(* IEC 61131-3 sources: open-ot-experiments/st/iec61131/tests, 28 files *)

(* ---- test_authoring_api.st ---- *)
FUNCTION OPENOT_AuthoringHeaderOk : BOOL
VAR_INPUT
    Records : OPENOT_SCAN_RECORD_BUFFER;
    Offset : UINT;
    Length : UINT;
    EventTypeId : UDINT;
    SourceId : UDINT;
END_VAR
VAR
    HeaderOk : BOOL;
    SourceRemaining : UDINT;
    EventRemaining : UDINT;
    Index : UINT;
    Pos : UINT;
END_VAR

HeaderOk :=
    (Length >= UINT#44) AND
    (Records[Offset] = BYTE#16#4F) AND
    (Records[Offset + UINT#1] = BYTE#16#4F) AND
    (Records[Offset + UINT#2] = BYTE#16#54) AND
    (Records[Offset + UINT#3] = BYTE#16#32) AND
    (Records[Offset + UINT#4] = UINT_TO_BYTE(Length MOD UINT#256)) AND
    (Records[Offset + UINT#5] = UINT_TO_BYTE((Length / UINT#256) MOD UINT#256)) AND
    (Records[Offset + UINT#6] = BYTE#16#08) AND
    (Records[Offset + UINT#7] = BYTE#16#00);

SourceRemaining := SourceId;
FOR Index := UINT#0 TO UINT#3 DO
    Pos := Offset + UINT#32 + Index;
    HeaderOk := HeaderOk AND (Records[Pos] = UDINT_TO_BYTE(SourceRemaining MOD UDINT#256));
    SourceRemaining := SourceRemaining / UDINT#256;
END_FOR;

EventRemaining := EventTypeId;
FOR Index := UINT#0 TO UINT#3 DO
    Pos := Offset + UINT#36 + Index;
    HeaderOk := HeaderOk AND (Records[Pos] = UDINT_TO_BYTE(EventRemaining MOD UDINT#256));
    EventRemaining := EventRemaining / UDINT#256;
END_FOR;

OPENOT_AuthoringHeaderOk := HeaderOk;
END_FUNCTION

FUNCTION_BLOCK OPENOT_TestAuthoringApi
VAR_OUTPUT
    Passed : BOOL;
    FirstBatchCount : UINT;
    FirstBatchDelta : ULINT;
    NoChangeCount : UINT;
    NoChangeDelta : ULINT;
    HeadersOk : BOOL;
    EmissionsOk : BOOL;
    ChangeSuppressionOk : BOOL;
END_VAR
VAR
    Producer : OPENOT_Producer;
    BeforeCount : ULINT;
    Offset0 : UINT;
    Offset1 : UINT;
    Offset2 : UINT;
    Length0 : UINT;
    Length1 : UINT;
    Length2 : UINT;
END_VAR

Producer(Execute := FALSE, ResetScanRecords := TRUE);
Producer(Execute := FALSE, ResetScanRecords := FALSE);
BeforeCount := Producer.PublishedRecordCount;
Producer(
    Execute := TRUE,
    Op := UINT#6,
    ValueId := UDINT#2001,
    ValueReal := REAL#12.5,
    DeadbandReal := REAL#0.5,
    HasQuality := FALSE,
    Quality := UINT#0);
Producer(Execute := FALSE, Op := UINT#6);
Producer(
    Execute := TRUE,
    Op := UINT#7,
    ValueId := UDINT#2002,
    ValueInt := DINT#42,
    HasQuality := FALSE,
    Quality := UINT#0);
Producer(Execute := FALSE, Op := UINT#7);
Producer(
    Execute := TRUE,
    Op := UINT#8,
    StateMachineId := UDINT#7,
    Category := UINT#2,
    PreviousState := UINT#0,
    NewState := UINT#1);
Producer(Execute := FALSE, Op := UINT#8);

FirstBatchCount := Producer.ScanRecordCount;
FirstBatchDelta := Producer.PublishedRecordCount - BeforeCount;
Offset0 := Producer.ScanRecordOffsets[0];
Offset1 := Producer.ScanRecordOffsets[1];
Offset2 := Producer.ScanRecordOffsets[2];
Length0 := Producer.ScanRecordLengths[0];
Length1 := Producer.ScanRecordLengths[1];
Length2 := Producer.ScanRecordLengths[2];
HeadersOk :=
    OPENOT_AuthoringHeaderOk(
        Records := Producer.ScanRecords,
        Offset := Offset0,
        Length := Length0,
        EventTypeId := UDINT#16#0002,
        SourceId := UDINT#1) AND
    OPENOT_AuthoringHeaderOk(
        Records := Producer.ScanRecords,
        Offset := Offset1,
        Length := Length1,
        EventTypeId := UDINT#16#0002,
        SourceId := UDINT#1) AND
    OPENOT_AuthoringHeaderOk(
        Records := Producer.ScanRecords,
        Offset := Offset2,
        Length := Length2,
        EventTypeId := UDINT#16#0001,
        SourceId := UDINT#1);

EmissionsOk :=
    (Producer.EmissionCount = UINT#3) AND
    (Producer.Emissions[0].EventTypeId = UDINT#16#0002) AND
    (Producer.Emissions[0].Seq = ULINT#0) AND
    (Producer.Emissions[1].EventTypeId = UDINT#16#0002) AND
    (Producer.Emissions[1].Seq = ULINT#1) AND
    (Producer.Emissions[2].EventTypeId = UDINT#16#0001) AND
    (Producer.Emissions[2].Seq = ULINT#2);

Producer(Execute := FALSE, ResetScanRecords := TRUE);
Producer(Execute := FALSE, ResetScanRecords := FALSE);
BeforeCount := Producer.PublishedRecordCount;
Producer(
    Execute := TRUE,
    Op := UINT#6,
    ValueId := UDINT#2001,
    ValueReal := REAL#12.5,
    DeadbandReal := REAL#0.5,
    HasQuality := FALSE,
    Quality := UINT#0);
Producer(Execute := FALSE, Op := UINT#6);
Producer(
    Execute := TRUE,
    Op := UINT#7,
    ValueId := UDINT#2002,
    ValueInt := DINT#42,
    HasQuality := FALSE,
    Quality := UINT#0);
Producer(Execute := FALSE, Op := UINT#7);
Producer(
    Execute := TRUE,
    Op := UINT#8,
    StateMachineId := UDINT#7,
    Category := UINT#2,
    PreviousState := UINT#0,
    NewState := UINT#1);
Producer(Execute := FALSE, Op := UINT#8);

NoChangeCount := Producer.ScanRecordCount;
NoChangeDelta := Producer.PublishedRecordCount - BeforeCount;
ChangeSuppressionOk := (NoChangeCount = UINT#0) AND (NoChangeDelta = ULINT#0);

Passed :=
    (FirstBatchCount = UINT#3) AND
    (FirstBatchDelta = ULINT#3) AND
    HeadersOk AND
    EmissionsOk AND
    ChangeSuppressionOk;
END_FUNCTION_BLOCK

(* ---- test_conformant_condition_lifecycle.st ---- *)
FUNCTION_BLOCK OPENOT_TestConformantConditionLifecycle
VAR_OUTPUT
    Passed : BOOL;
    AckPassed : BOOL;
    ShelvedPassed : BOOL;
    SuppressedPassed : BOOL;
    OutOfServicePassed : BOOL;
    MismatchIndex : UINT;
END_VAR
VAR
    AckEncoder : OPENOT_EncodeConformantConditionAcknowledged;
    ShelvedEncoder : OPENOT_EncodeConformantConditionShelved;
    SuppressedEncoder : OPENOT_EncodeConformantConditionSuppressed;
    OutOfServiceEncoder : OPENOT_EncodeConformantConditionOutOfService;
    ExpectedAck : ARRAY[0..75] OF BYTE := [
        BYTE#16#4F, BYTE#16#4F, BYTE#16#54, BYTE#16#32, BYTE#16#4C, BYTE#16#00, BYTE#16#08, BYTE#16#00,
        BYTE#16#A0, BYTE#16#CA, BYTE#16#9A, BYTE#16#3B, BYTE#16#00, BYTE#16#00, BYTE#16#00, BYTE#16#00,
        BYTE#16#01, BYTE#16#00, BYTE#16#00, BYTE#16#00, BYTE#16#00, BYTE#16#00, BYTE#16#00, BYTE#16#00,
        BYTE#16#11, BYTE#16#00, BYTE#16#00, BYTE#16#00, BYTE#16#00, BYTE#16#00, BYTE#16#00, BYTE#16#00,
        BYTE#16#42, BYTE#16#00, BYTE#16#00, BYTE#16#00, BYTE#16#02, BYTE#16#02, BYTE#16#00, BYTE#16#00,
        BYTE#16#05, BYTE#16#00, BYTE#16#05, BYTE#16#04, BYTE#16#29, BYTE#16#23, BYTE#16#00, BYTE#16#00,
        BYTE#16#07, BYTE#16#00, BYTE#16#05, BYTE#16#04, BYTE#16#4D, BYTE#16#00, BYTE#16#00, BYTE#16#00,
        BYTE#16#1D, BYTE#16#00, BYTE#16#0C, BYTE#16#0A, BYTE#16#6F, BYTE#16#70, BYTE#16#65, BYTE#16#72,
        BYTE#16#61, BYTE#16#74, BYTE#16#6F, BYTE#16#72, BYTE#16#2D, BYTE#16#61, BYTE#16#00, BYTE#16#00,
        BYTE#16#FA, BYTE#16#EA, BYTE#16#82, BYTE#16#EC
    ];
    ExpectedShelved : ARRAY[0..83] OF BYTE := [
        BYTE#16#4F, BYTE#16#4F, BYTE#16#54, BYTE#16#32, BYTE#16#54, BYTE#16#00, BYTE#16#08, BYTE#16#00,
        BYTE#16#AA, BYTE#16#CA, BYTE#16#9A, BYTE#16#3B, BYTE#16#00, BYTE#16#00, BYTE#16#00, BYTE#16#00,
        BYTE#16#01, BYTE#16#00, BYTE#16#00, BYTE#16#00, BYTE#16#00, BYTE#16#00, BYTE#16#00, BYTE#16#00,
        BYTE#16#12, BYTE#16#00, BYTE#16#00, BYTE#16#00, BYTE#16#00, BYTE#16#00, BYTE#16#00, BYTE#16#00,
        BYTE#16#42, BYTE#16#00, BYTE#16#00, BYTE#16#00, BYTE#16#04, BYTE#16#02, BYTE#16#00, BYTE#16#00,
        BYTE#16#05, BYTE#16#00, BYTE#16#05, BYTE#16#04, BYTE#16#29, BYTE#16#23, BYTE#16#00, BYTE#16#00,
        BYTE#16#07, BYTE#16#00, BYTE#16#05, BYTE#16#04, BYTE#16#4D, BYTE#16#00, BYTE#16#00, BYTE#16#00,
        BYTE#16#1D, BYTE#16#00, BYTE#16#0C, BYTE#16#0A, BYTE#16#6F, BYTE#16#70, BYTE#16#65, BYTE#16#72,
        BYTE#16#61, BYTE#16#74, BYTE#16#6F, BYTE#16#72, BYTE#16#2D, BYTE#16#61, BYTE#16#00, BYTE#16#00,
        BYTE#16#1E, BYTE#16#00, BYTE#16#05, BYTE#16#04, BYTE#16#2C, BYTE#16#01, BYTE#16#00, BYTE#16#00,
        BYTE#16#E5, BYTE#16#3E, BYTE#16#92, BYTE#16#BD
    ];
    ExpectedSuppressed : ARRAY[0..67] OF BYTE := [
        BYTE#16#4F, BYTE#16#4F, BYTE#16#54, BYTE#16#32, BYTE#16#44, BYTE#16#00, BYTE#16#08, BYTE#16#00,
        BYTE#16#B4, BYTE#16#CA, BYTE#16#9A, BYTE#16#3B, BYTE#16#00, BYTE#16#00, BYTE#16#00, BYTE#16#00,
        BYTE#16#01, BYTE#16#00, BYTE#16#00, BYTE#16#00, BYTE#16#00, BYTE#16#00, BYTE#16#00, BYTE#16#00,
        BYTE#16#13, BYTE#16#00, BYTE#16#00, BYTE#16#00, BYTE#16#00, BYTE#16#00, BYTE#16#00, BYTE#16#00,
        BYTE#16#42, BYTE#16#00, BYTE#16#00, BYTE#16#00, BYTE#16#06, BYTE#16#02, BYTE#16#00, BYTE#16#00,
        BYTE#16#05, BYTE#16#00, BYTE#16#05, BYTE#16#04, BYTE#16#29, BYTE#16#23, BYTE#16#00, BYTE#16#00,
        BYTE#16#1F, BYTE#16#00, BYTE#16#0C, BYTE#16#0B, BYTE#16#6D, BYTE#16#61, BYTE#16#69, BYTE#16#6E,
        BYTE#16#74, BYTE#16#65, BYTE#16#6E, BYTE#16#61, BYTE#16#6E, BYTE#16#63, BYTE#16#65, BYTE#16#00,
        BYTE#16#17, BYTE#16#3E, BYTE#16#4F, BYTE#16#63
    ];
    ExpectedOutOfService : ARRAY[0..67] OF BYTE := [
        BYTE#16#4F, BYTE#16#4F, BYTE#16#54, BYTE#16#32, BYTE#16#44, BYTE#16#00, BYTE#16#08, BYTE#16#00,
        BYTE#16#BE, BYTE#16#CA, BYTE#16#9A, BYTE#16#3B, BYTE#16#00, BYTE#16#00, BYTE#16#00, BYTE#16#00,
        BYTE#16#01, BYTE#16#00, BYTE#16#00, BYTE#16#00, BYTE#16#00, BYTE#16#00, BYTE#16#00, BYTE#16#00,
        BYTE#16#14, BYTE#16#00, BYTE#16#00, BYTE#16#00, BYTE#16#00, BYTE#16#00, BYTE#16#00, BYTE#16#00,
        BYTE#16#42, BYTE#16#00, BYTE#16#00, BYTE#16#00, BYTE#16#08, BYTE#16#02, BYTE#16#00, BYTE#16#00,
        BYTE#16#05, BYTE#16#00, BYTE#16#05, BYTE#16#04, BYTE#16#29, BYTE#16#23, BYTE#16#00, BYTE#16#00,
        BYTE#16#1D, BYTE#16#00, BYTE#16#0C, BYTE#16#0A, BYTE#16#6F, BYTE#16#70, BYTE#16#65, BYTE#16#72,
        BYTE#16#61, BYTE#16#74, BYTE#16#6F, BYTE#16#72, BYTE#16#2D, BYTE#16#61, BYTE#16#00, BYTE#16#00,
        BYTE#16#9D, BYTE#16#5C, BYTE#16#A4, BYTE#16#01
    ];
    Index : UINT;
END_VAR

AckEncoder();
ShelvedEncoder();
SuppressedEncoder();
OutOfServiceEncoder();

AckPassed := AckEncoder.Length = UINT#76;
ShelvedPassed := ShelvedEncoder.Length = UINT#84;
SuppressedPassed := SuppressedEncoder.Length = UINT#68;
OutOfServicePassed := OutOfServiceEncoder.Length = UINT#68;
MismatchIndex := UINT#65535;

IF AckPassed THEN
    FOR Index := UINT#0 TO UINT#75 DO
        IF (AckEncoder.Buffer[Index] <> ExpectedAck[Index]) AND (MismatchIndex = UINT#65535) THEN
            AckPassed := FALSE;
            MismatchIndex := Index;
        END_IF;
    END_FOR;
END_IF;

IF ShelvedPassed THEN
    FOR Index := UINT#0 TO UINT#83 DO
        IF (ShelvedEncoder.Buffer[Index] <> ExpectedShelved[Index]) AND (MismatchIndex = UINT#65535) THEN
            ShelvedPassed := FALSE;
            MismatchIndex := Index;
        END_IF;
    END_FOR;
END_IF;

IF SuppressedPassed THEN
    FOR Index := UINT#0 TO UINT#67 DO
        IF (SuppressedEncoder.Buffer[Index] <> ExpectedSuppressed[Index]) AND (MismatchIndex = UINT#65535) THEN
            SuppressedPassed := FALSE;
            MismatchIndex := Index;
        END_IF;
    END_FOR;
END_IF;

IF OutOfServicePassed THEN
    FOR Index := UINT#0 TO UINT#67 DO
        IF (OutOfServiceEncoder.Buffer[Index] <> ExpectedOutOfService[Index]) AND (MismatchIndex = UINT#65535) THEN
            OutOfServicePassed := FALSE;
            MismatchIndex := Index;
        END_IF;
    END_FOR;
END_IF;

Passed := AckPassed AND ShelvedPassed AND SuppressedPassed AND OutOfServicePassed;
END_FUNCTION_BLOCK

(* ---- test_conformant_message.st ---- *)
FUNCTION_BLOCK OPENOT_TestConformantMessage
VAR_OUTPUT
    Passed : BOOL;
    MismatchIndex : UINT;
    ActualLength : UINT;
    ExpectedLength : UINT;
END_VAR
VAR
    Encoder : OPENOT_EncodeConformantMessage;
    Expected : ARRAY[0..75] OF BYTE := [
        BYTE#16#4F, BYTE#16#4F, BYTE#16#54, BYTE#16#32, BYTE#16#4C, BYTE#16#00, BYTE#16#08, BYTE#16#00,
        BYTE#16#0A, BYTE#16#CA, BYTE#16#9A, BYTE#16#3B, BYTE#16#00, BYTE#16#00, BYTE#16#00, BYTE#16#00,
        BYTE#16#01, BYTE#16#00, BYTE#16#00, BYTE#16#00, BYTE#16#00, BYTE#16#00, BYTE#16#00, BYTE#16#00,
        BYTE#16#02, BYTE#16#00, BYTE#16#00, BYTE#16#00, BYTE#16#00, BYTE#16#00, BYTE#16#00, BYTE#16#00,
        BYTE#16#42, BYTE#16#00, BYTE#16#00, BYTE#16#00, BYTE#16#03, BYTE#16#00, BYTE#16#00, BYTE#16#00,
        BYTE#16#14, BYTE#16#00, BYTE#16#05, BYTE#16#04, BYTE#16#E9, BYTE#16#03, BYTE#16#00, BYTE#16#00,
        BYTE#16#15, BYTE#16#00, BYTE#16#0C, BYTE#16#0B, BYTE#16#70, BYTE#16#68, BYTE#16#61, BYTE#16#73,
        BYTE#16#65, BYTE#16#20, BYTE#16#72, BYTE#16#65, BYTE#16#61, BYTE#16#64, BYTE#16#79, BYTE#16#00,
        BYTE#16#08, BYTE#16#00, BYTE#16#03, BYTE#16#02, BYTE#16#F4, BYTE#16#01, BYTE#16#00, BYTE#16#00,
        BYTE#16#CF, BYTE#16#CF, BYTE#16#BE, BYTE#16#B0
    ];
    Index : UINT;
END_VAR

Encoder();
ActualLength := Encoder.Length;
ExpectedLength := UINT#76;
Passed := ActualLength = ExpectedLength;
MismatchIndex := UINT#65535;

IF Passed THEN
    FOR Index := UINT#0 TO ExpectedLength - UINT#1 DO
        IF (Encoder.Buffer[Index] <> Expected[Index]) AND (MismatchIndex = UINT#65535) THEN
            Passed := FALSE;
            MismatchIndex := Index;
        END_IF;
    END_FOR;
END_IF;
END_FUNCTION_BLOCK

(* ---- test_conformant_records_dropped.st ---- *)
FUNCTION_BLOCK OPENOT_TestConformantRecordsDropped
VAR_OUTPUT
    Passed : BOOL;
    MismatchIndex : UINT;
    ActualLength : UINT;
    ExpectedLength : UINT;
END_VAR
VAR
    Encoder : OPENOT_EncodeConformantRecordsDropped;
    Expected : ARRAY[0..99] OF BYTE := [
        BYTE#16#4F, BYTE#16#4F, BYTE#16#54, BYTE#16#32, BYTE#16#64, BYTE#16#00, BYTE#16#08, BYTE#16#00,
        BYTE#16#00, BYTE#16#00, BYTE#16#00, BYTE#16#00, BYTE#16#00, BYTE#16#00, BYTE#16#00, BYTE#16#00,
        BYTE#16#09, BYTE#16#00, BYTE#16#00, BYTE#16#00, BYTE#16#00, BYTE#16#00, BYTE#16#00, BYTE#16#00,
        BYTE#16#64, BYTE#16#00, BYTE#16#00, BYTE#16#00, BYTE#16#00, BYTE#16#00, BYTE#16#00, BYTE#16#00,
        BYTE#16#42, BYTE#16#00, BYTE#16#00, BYTE#16#00, BYTE#16#04, BYTE#16#01, BYTE#16#00, BYTE#16#00,
        BYTE#16#16, BYTE#16#00, BYTE#16#05, BYTE#16#04, BYTE#16#12, BYTE#16#00, BYTE#16#00, BYTE#16#00,
        BYTE#16#17, BYTE#16#00, BYTE#16#07, BYTE#16#08, BYTE#16#28, BYTE#16#00, BYTE#16#00, BYTE#16#00,
        BYTE#16#00, BYTE#16#00, BYTE#16#00, BYTE#16#00, BYTE#16#18, BYTE#16#00, BYTE#16#07, BYTE#16#08,
        BYTE#16#39, BYTE#16#00, BYTE#16#00, BYTE#16#00, BYTE#16#00, BYTE#16#00, BYTE#16#00, BYTE#16#00,
        BYTE#16#19, BYTE#16#00, BYTE#16#0B, BYTE#16#08, BYTE#16#00, BYTE#16#CA, BYTE#16#9A, BYTE#16#3B,
        BYTE#16#00, BYTE#16#00, BYTE#16#00, BYTE#16#00, BYTE#16#1A, BYTE#16#00, BYTE#16#0B, BYTE#16#08,
        BYTE#16#10, BYTE#16#F1, BYTE#16#9A, BYTE#16#3B, BYTE#16#00, BYTE#16#00, BYTE#16#00, BYTE#16#00,
        BYTE#16#09, BYTE#16#8A, BYTE#16#DF, BYTE#16#6D
    ];
    Index : UINT;
END_VAR

Encoder();
ActualLength := Encoder.Length;
ExpectedLength := UINT#100;
Passed := ActualLength = ExpectedLength;
MismatchIndex := UINT#65535;

IF Passed THEN
    FOR Index := UINT#0 TO ExpectedLength - UINT#1 DO
        IF (Encoder.Buffer[Index] <> Expected[Index]) AND (MismatchIndex = UINT#65535) THEN
            Passed := FALSE;
            MismatchIndex := Index;
        END_IF;
    END_FOR;
END_IF;
END_FUNCTION_BLOCK

(* ---- test_conformant_regulated.st ---- *)
FUNCTION_BLOCK OPENOT_TestConformantRegulated
VAR_OUTPUT
    Passed : BOOL;
    OperatorActionPassed : BOOL;
    OperatorLoginPassed : BOOL;
    OperatorLogoutPassed : BOOL;
    SecurityAccessFailurePassed : BOOL;
    ParameterChangeRealPassed : BOOL;
    ParameterChangeIntPassed : BOOL;
    ParameterChangeBitsPassed : BOOL;
    ParameterChangeStringPassed : BOOL;
    MismatchIndex : UINT;
END_VAR
VAR
    OperatorActionEncoder : OPENOT_EncodeConformantOperatorAction;
    OperatorLoginEncoder : OPENOT_EncodeConformantOperatorLogin;
    OperatorLogoutEncoder : OPENOT_EncodeConformantOperatorLogout;
    SecurityAccessFailureEncoder : OPENOT_EncodeConformantSecurityAccessFailure;
    ParameterChangeRealEncoder : OPENOT_EncodeConformantParameterChangeReal;
    ParameterChangeIntEncoder : OPENOT_EncodeConformantParameterChangeInt;
    ParameterChangeBitsEncoder : OPENOT_EncodeConformantParameterChangeBits;
    ParameterChangeStringEncoder : OPENOT_EncodeConformantParameterChangeString;
    ExpectedOperatorAction : ARRAY[0..107] OF BYTE := [
        BYTE#16#4F, BYTE#16#4F, BYTE#16#54, BYTE#16#32, BYTE#16#6C, BYTE#16#00, BYTE#16#08, BYTE#16#00, BYTE#16#36, BYTE#16#CB, BYTE#16#9A, BYTE#16#3B, BYTE#16#00, BYTE#16#00, BYTE#16#00, BYTE#16#00,
        BYTE#16#01, BYTE#16#00, BYTE#16#00, BYTE#16#00, BYTE#16#00, BYTE#16#00, BYTE#16#00, BYTE#16#00, BYTE#16#20, BYTE#16#00, BYTE#16#00, BYTE#16#00, BYTE#16#00, BYTE#16#00, BYTE#16#00, BYTE#16#00,
        BYTE#16#42, BYTE#16#00, BYTE#16#00, BYTE#16#00, BYTE#16#00, BYTE#16#04, BYTE#16#00, BYTE#16#00, BYTE#16#0A, BYTE#16#00, BYTE#16#05, BYTE#16#04, BYTE#16#71, BYTE#16#17, BYTE#16#00, BYTE#16#00,
        BYTE#16#0B, BYTE#16#00, BYTE#16#0C, BYTE#16#0A, BYTE#16#6F, BYTE#16#70, BYTE#16#65, BYTE#16#72, BYTE#16#61, BYTE#16#74, BYTE#16#6F, BYTE#16#72, BYTE#16#2D, BYTE#16#61, BYTE#16#00, BYTE#16#00,
        BYTE#16#0C, BYTE#16#00, BYTE#16#05, BYTE#16#04, BYTE#16#59, BYTE#16#1B, BYTE#16#00, BYTE#16#00, BYTE#16#0C, BYTE#16#00, BYTE#16#05, BYTE#16#04, BYTE#16#5A, BYTE#16#1B, BYTE#16#00, BYTE#16#00,
        BYTE#16#20, BYTE#16#00, BYTE#16#03, BYTE#16#02, BYTE#16#00, BYTE#16#00, BYTE#16#00, BYTE#16#00, BYTE#16#21, BYTE#16#00, BYTE#16#0C, BYTE#16#09, BYTE#16#73, BYTE#16#74, BYTE#16#61, BYTE#16#74,
        BYTE#16#69, BYTE#16#6F, BYTE#16#6E, BYTE#16#2D, BYTE#16#31, BYTE#16#00, BYTE#16#00, BYTE#16#00, BYTE#16#26, BYTE#16#B1, BYTE#16#DF, BYTE#16#49
    ];
    ExpectedOperatorLogin : ARRAY[0..91] OF BYTE := [
        BYTE#16#4F, BYTE#16#4F, BYTE#16#54, BYTE#16#32, BYTE#16#5C, BYTE#16#00, BYTE#16#08, BYTE#16#00, BYTE#16#40, BYTE#16#CB, BYTE#16#9A, BYTE#16#3B, BYTE#16#00, BYTE#16#00, BYTE#16#00, BYTE#16#00,
        BYTE#16#01, BYTE#16#00, BYTE#16#00, BYTE#16#00, BYTE#16#00, BYTE#16#00, BYTE#16#00, BYTE#16#00, BYTE#16#21, BYTE#16#00, BYTE#16#00, BYTE#16#00, BYTE#16#00, BYTE#16#00, BYTE#16#00, BYTE#16#00,
        BYTE#16#42, BYTE#16#00, BYTE#16#00, BYTE#16#00, BYTE#16#01, BYTE#16#04, BYTE#16#00, BYTE#16#00, BYTE#16#0B, BYTE#16#00, BYTE#16#0C, BYTE#16#0A, BYTE#16#6F, BYTE#16#70, BYTE#16#65, BYTE#16#72,
        BYTE#16#61, BYTE#16#74, BYTE#16#6F, BYTE#16#72, BYTE#16#2D, BYTE#16#61, BYTE#16#00, BYTE#16#00, BYTE#16#20, BYTE#16#00, BYTE#16#03, BYTE#16#02, BYTE#16#00, BYTE#16#00, BYTE#16#00, BYTE#16#00,
        BYTE#16#21, BYTE#16#00, BYTE#16#0C, BYTE#16#09, BYTE#16#73, BYTE#16#74, BYTE#16#61, BYTE#16#74, BYTE#16#69, BYTE#16#6F, BYTE#16#6E, BYTE#16#2D, BYTE#16#31, BYTE#16#00, BYTE#16#00, BYTE#16#00,
        BYTE#16#33, BYTE#16#00, BYTE#16#03, BYTE#16#02, BYTE#16#03, BYTE#16#00, BYTE#16#00, BYTE#16#00, BYTE#16#74, BYTE#16#13, BYTE#16#41, BYTE#16#A8
    ];
    ExpectedOperatorLogout : ARRAY[0..75] OF BYTE := [
        BYTE#16#4F, BYTE#16#4F, BYTE#16#54, BYTE#16#32, BYTE#16#4C, BYTE#16#00, BYTE#16#08, BYTE#16#00, BYTE#16#4A, BYTE#16#CB, BYTE#16#9A, BYTE#16#3B, BYTE#16#00, BYTE#16#00, BYTE#16#00, BYTE#16#00,
        BYTE#16#01, BYTE#16#00, BYTE#16#00, BYTE#16#00, BYTE#16#00, BYTE#16#00, BYTE#16#00, BYTE#16#00, BYTE#16#22, BYTE#16#00, BYTE#16#00, BYTE#16#00, BYTE#16#00, BYTE#16#00, BYTE#16#00, BYTE#16#00,
        BYTE#16#42, BYTE#16#00, BYTE#16#00, BYTE#16#00, BYTE#16#02, BYTE#16#04, BYTE#16#00, BYTE#16#00, BYTE#16#0B, BYTE#16#00, BYTE#16#0C, BYTE#16#0A, BYTE#16#6F, BYTE#16#70, BYTE#16#65, BYTE#16#72,
        BYTE#16#61, BYTE#16#74, BYTE#16#6F, BYTE#16#72, BYTE#16#2D, BYTE#16#61, BYTE#16#00, BYTE#16#00, BYTE#16#21, BYTE#16#00, BYTE#16#0C, BYTE#16#09, BYTE#16#73, BYTE#16#74, BYTE#16#61, BYTE#16#74,
        BYTE#16#69, BYTE#16#6F, BYTE#16#6E, BYTE#16#2D, BYTE#16#31, BYTE#16#00, BYTE#16#00, BYTE#16#00, BYTE#16#14, BYTE#16#BF, BYTE#16#E7, BYTE#16#8C
    ];
    ExpectedSecurityAccessFailure : ARRAY[0..87] OF BYTE := [
        BYTE#16#4F, BYTE#16#4F, BYTE#16#54, BYTE#16#32, BYTE#16#58, BYTE#16#00, BYTE#16#08, BYTE#16#00, BYTE#16#54, BYTE#16#CB, BYTE#16#9A, BYTE#16#3B, BYTE#16#00, BYTE#16#00, BYTE#16#00, BYTE#16#00,
        BYTE#16#01, BYTE#16#00, BYTE#16#00, BYTE#16#00, BYTE#16#00, BYTE#16#00, BYTE#16#00, BYTE#16#00, BYTE#16#23, BYTE#16#00, BYTE#16#00, BYTE#16#00, BYTE#16#00, BYTE#16#00, BYTE#16#00, BYTE#16#00,
        BYTE#16#42, BYTE#16#00, BYTE#16#00, BYTE#16#00, BYTE#16#05, BYTE#16#04, BYTE#16#00, BYTE#16#00, BYTE#16#0B, BYTE#16#00, BYTE#16#0C, BYTE#16#0A, BYTE#16#6F, BYTE#16#70, BYTE#16#65, BYTE#16#72,
        BYTE#16#61, BYTE#16#74, BYTE#16#6F, BYTE#16#72, BYTE#16#2D, BYTE#16#78, BYTE#16#00, BYTE#16#00, BYTE#16#21, BYTE#16#00, BYTE#16#0C, BYTE#16#09, BYTE#16#73, BYTE#16#74, BYTE#16#61, BYTE#16#74,
        BYTE#16#69, BYTE#16#6F, BYTE#16#6E, BYTE#16#2D, BYTE#16#32, BYTE#16#00, BYTE#16#00, BYTE#16#00, BYTE#16#1F, BYTE#16#00, BYTE#16#0C, BYTE#16#06, BYTE#16#64, BYTE#16#65, BYTE#16#6E, BYTE#16#69,
        BYTE#16#65, BYTE#16#64, BYTE#16#00, BYTE#16#00, BYTE#16#47, BYTE#16#D1, BYTE#16#30, BYTE#16#F7
    ];
    ExpectedParameterChangeReal : ARRAY[0..111] OF BYTE := [
        BYTE#16#4F, BYTE#16#4F, BYTE#16#54, BYTE#16#32, BYTE#16#70, BYTE#16#00, BYTE#16#08, BYTE#16#00, BYTE#16#5E, BYTE#16#CB, BYTE#16#9A, BYTE#16#3B, BYTE#16#00, BYTE#16#00, BYTE#16#00, BYTE#16#00,
        BYTE#16#01, BYTE#16#00, BYTE#16#00, BYTE#16#00, BYTE#16#00, BYTE#16#00, BYTE#16#00, BYTE#16#00, BYTE#16#24, BYTE#16#00, BYTE#16#00, BYTE#16#00, BYTE#16#00, BYTE#16#00, BYTE#16#00, BYTE#16#00,
        BYTE#16#42, BYTE#16#00, BYTE#16#00, BYTE#16#00, BYTE#16#03, BYTE#16#04, BYTE#16#00, BYTE#16#00, BYTE#16#0D, BYTE#16#00, BYTE#16#05, BYTE#16#04, BYTE#16#D1, BYTE#16#07, BYTE#16#00, BYTE#16#00,
        BYTE#16#0F, BYTE#16#00, BYTE#16#09, BYTE#16#04, BYTE#16#00, BYTE#16#00, BYTE#16#48, BYTE#16#41, BYTE#16#10, BYTE#16#00, BYTE#16#09, BYTE#16#04, BYTE#16#00, BYTE#16#00, BYTE#16#5C, BYTE#16#41,
        BYTE#16#0B, BYTE#16#00, BYTE#16#0C, BYTE#16#0A, BYTE#16#6F, BYTE#16#70, BYTE#16#65, BYTE#16#72, BYTE#16#61, BYTE#16#74, BYTE#16#6F, BYTE#16#72, BYTE#16#2D, BYTE#16#61, BYTE#16#00, BYTE#16#00,
        BYTE#16#1F, BYTE#16#00, BYTE#16#0C, BYTE#16#0F, BYTE#16#73, BYTE#16#65, BYTE#16#74, BYTE#16#70, BYTE#16#6F, BYTE#16#69, BYTE#16#6E, BYTE#16#74, BYTE#16#20, BYTE#16#63, BYTE#16#68, BYTE#16#61,
        BYTE#16#6E, BYTE#16#67, BYTE#16#65, BYTE#16#00, BYTE#16#20, BYTE#16#00, BYTE#16#03, BYTE#16#02, BYTE#16#00, BYTE#16#00, BYTE#16#00, BYTE#16#00, BYTE#16#C6, BYTE#16#34, BYTE#16#40, BYTE#16#11
    ];
    ExpectedParameterChangeInt : ARRAY[0..103] OF BYTE := [
        BYTE#16#4F, BYTE#16#4F, BYTE#16#54, BYTE#16#32, BYTE#16#68, BYTE#16#00, BYTE#16#08, BYTE#16#00, BYTE#16#68, BYTE#16#CB, BYTE#16#9A, BYTE#16#3B, BYTE#16#00, BYTE#16#00, BYTE#16#00, BYTE#16#00,
        BYTE#16#01, BYTE#16#00, BYTE#16#00, BYTE#16#00, BYTE#16#00, BYTE#16#00, BYTE#16#00, BYTE#16#00, BYTE#16#25, BYTE#16#00, BYTE#16#00, BYTE#16#00, BYTE#16#00, BYTE#16#00, BYTE#16#00, BYTE#16#00,
        BYTE#16#42, BYTE#16#00, BYTE#16#00, BYTE#16#00, BYTE#16#03, BYTE#16#04, BYTE#16#00, BYTE#16#00, BYTE#16#0D, BYTE#16#00, BYTE#16#05, BYTE#16#04, BYTE#16#D2, BYTE#16#07, BYTE#16#00, BYTE#16#00,
        BYTE#16#0F, BYTE#16#00, BYTE#16#06, BYTE#16#04, BYTE#16#28, BYTE#16#00, BYTE#16#00, BYTE#16#00, BYTE#16#10, BYTE#16#00, BYTE#16#06, BYTE#16#04, BYTE#16#2A, BYTE#16#00, BYTE#16#00, BYTE#16#00,
        BYTE#16#0B, BYTE#16#00, BYTE#16#0C, BYTE#16#0A, BYTE#16#6F, BYTE#16#70, BYTE#16#65, BYTE#16#72, BYTE#16#61, BYTE#16#74, BYTE#16#6F, BYTE#16#72, BYTE#16#2D, BYTE#16#61, BYTE#16#00, BYTE#16#00,
        BYTE#16#1F, BYTE#16#00, BYTE#16#0C, BYTE#16#0F, BYTE#16#63, BYTE#16#6F, BYTE#16#75, BYTE#16#6E, BYTE#16#74, BYTE#16#20, BYTE#16#63, BYTE#16#6F, BYTE#16#72, BYTE#16#72, BYTE#16#65, BYTE#16#63,
        BYTE#16#74, BYTE#16#65, BYTE#16#64, BYTE#16#00, BYTE#16#7F, BYTE#16#51, BYTE#16#5C, BYTE#16#9A
    ];
    ExpectedParameterChangeBits : ARRAY[0..99] OF BYTE := [
        BYTE#16#4F, BYTE#16#4F, BYTE#16#54, BYTE#16#32, BYTE#16#64, BYTE#16#00, BYTE#16#08, BYTE#16#00, BYTE#16#72, BYTE#16#CB, BYTE#16#9A, BYTE#16#3B, BYTE#16#00, BYTE#16#00, BYTE#16#00, BYTE#16#00,
        BYTE#16#01, BYTE#16#00, BYTE#16#00, BYTE#16#00, BYTE#16#00, BYTE#16#00, BYTE#16#00, BYTE#16#00, BYTE#16#26, BYTE#16#00, BYTE#16#00, BYTE#16#00, BYTE#16#00, BYTE#16#00, BYTE#16#00, BYTE#16#00,
        BYTE#16#42, BYTE#16#00, BYTE#16#00, BYTE#16#00, BYTE#16#03, BYTE#16#04, BYTE#16#00, BYTE#16#00, BYTE#16#0D, BYTE#16#00, BYTE#16#05, BYTE#16#04, BYTE#16#D3, BYTE#16#07, BYTE#16#00, BYTE#16#00,
        BYTE#16#0F, BYTE#16#00, BYTE#16#00, BYTE#16#01, BYTE#16#00, BYTE#16#00, BYTE#16#00, BYTE#16#00, BYTE#16#10, BYTE#16#00, BYTE#16#00, BYTE#16#01, BYTE#16#01, BYTE#16#00, BYTE#16#00, BYTE#16#00,
        BYTE#16#0B, BYTE#16#00, BYTE#16#0C, BYTE#16#0A, BYTE#16#6F, BYTE#16#70, BYTE#16#65, BYTE#16#72, BYTE#16#61, BYTE#16#74, BYTE#16#6F, BYTE#16#72, BYTE#16#2D, BYTE#16#62, BYTE#16#00, BYTE#16#00,
        BYTE#16#1F, BYTE#16#00, BYTE#16#0C, BYTE#16#0C, BYTE#16#65, BYTE#16#6E, BYTE#16#61, BYTE#16#62, BYTE#16#6C, BYTE#16#65, BYTE#16#20, BYTE#16#61, BYTE#16#75, BYTE#16#64, BYTE#16#69, BYTE#16#74,
        BYTE#16#59, BYTE#16#CA, BYTE#16#6A, BYTE#16#6E
    ];
    ExpectedParameterChangeString : ARRAY[0..111] OF BYTE := [
        BYTE#16#4F, BYTE#16#4F, BYTE#16#54, BYTE#16#32, BYTE#16#70, BYTE#16#00, BYTE#16#08, BYTE#16#00, BYTE#16#7C, BYTE#16#CB, BYTE#16#9A, BYTE#16#3B, BYTE#16#00, BYTE#16#00, BYTE#16#00, BYTE#16#00,
        BYTE#16#01, BYTE#16#00, BYTE#16#00, BYTE#16#00, BYTE#16#00, BYTE#16#00, BYTE#16#00, BYTE#16#00, BYTE#16#27, BYTE#16#00, BYTE#16#00, BYTE#16#00, BYTE#16#00, BYTE#16#00, BYTE#16#00, BYTE#16#00,
        BYTE#16#42, BYTE#16#00, BYTE#16#00, BYTE#16#00, BYTE#16#03, BYTE#16#04, BYTE#16#00, BYTE#16#00, BYTE#16#0D, BYTE#16#00, BYTE#16#05, BYTE#16#04, BYTE#16#DC, BYTE#16#07, BYTE#16#00, BYTE#16#00,
        BYTE#16#0F, BYTE#16#00, BYTE#16#0C, BYTE#16#06, BYTE#16#6D, BYTE#16#61, BYTE#16#6E, BYTE#16#75, BYTE#16#61, BYTE#16#6C, BYTE#16#00, BYTE#16#00, BYTE#16#10, BYTE#16#00, BYTE#16#0C, BYTE#16#04,
        BYTE#16#61, BYTE#16#75, BYTE#16#74, BYTE#16#6F, BYTE#16#0B, BYTE#16#00, BYTE#16#0C, BYTE#16#0A, BYTE#16#6F, BYTE#16#70, BYTE#16#65, BYTE#16#72, BYTE#16#61, BYTE#16#74, BYTE#16#6F, BYTE#16#72,
        BYTE#16#2D, BYTE#16#63, BYTE#16#00, BYTE#16#00, BYTE#16#1F, BYTE#16#00, BYTE#16#0C, BYTE#16#09, BYTE#16#6D, BYTE#16#6F, BYTE#16#64, BYTE#16#65, BYTE#16#20, BYTE#16#6E, BYTE#16#6F, BYTE#16#74,
        BYTE#16#65, BYTE#16#00, BYTE#16#00, BYTE#16#00, BYTE#16#20, BYTE#16#00, BYTE#16#03, BYTE#16#02, BYTE#16#01, BYTE#16#00, BYTE#16#00, BYTE#16#00, BYTE#16#76, BYTE#16#BE, BYTE#16#68, BYTE#16#A4
    ];
    Index : UINT;
END_VAR

OperatorActionEncoder();
OperatorLoginEncoder();
OperatorLogoutEncoder();
SecurityAccessFailureEncoder();
ParameterChangeRealEncoder();
ParameterChangeIntEncoder();
ParameterChangeBitsEncoder();
ParameterChangeStringEncoder();

OperatorActionPassed := OperatorActionEncoder.Length = UINT#108;
OperatorLoginPassed := OperatorLoginEncoder.Length = UINT#92;
OperatorLogoutPassed := OperatorLogoutEncoder.Length = UINT#76;
SecurityAccessFailurePassed := SecurityAccessFailureEncoder.Length = UINT#88;
ParameterChangeRealPassed := ParameterChangeRealEncoder.Length = UINT#112;
ParameterChangeIntPassed := ParameterChangeIntEncoder.Length = UINT#104;
ParameterChangeBitsPassed := ParameterChangeBitsEncoder.Length = UINT#100;
ParameterChangeStringPassed := ParameterChangeStringEncoder.Length = UINT#112;
MismatchIndex := UINT#65535;

IF OperatorActionPassed THEN
    FOR Index := UINT#0 TO UINT#107 DO
        IF (OperatorActionEncoder.Buffer[Index] <> ExpectedOperatorAction[Index]) AND (MismatchIndex = UINT#65535) THEN
            OperatorActionPassed := FALSE;
            MismatchIndex := Index;
        END_IF;
    END_FOR;
END_IF;

IF OperatorLoginPassed THEN
    FOR Index := UINT#0 TO UINT#91 DO
        IF (OperatorLoginEncoder.Buffer[Index] <> ExpectedOperatorLogin[Index]) AND (MismatchIndex = UINT#65535) THEN
            OperatorLoginPassed := FALSE;
            MismatchIndex := Index;
        END_IF;
    END_FOR;
END_IF;

IF OperatorLogoutPassed THEN
    FOR Index := UINT#0 TO UINT#75 DO
        IF (OperatorLogoutEncoder.Buffer[Index] <> ExpectedOperatorLogout[Index]) AND (MismatchIndex = UINT#65535) THEN
            OperatorLogoutPassed := FALSE;
            MismatchIndex := Index;
        END_IF;
    END_FOR;
END_IF;

IF SecurityAccessFailurePassed THEN
    FOR Index := UINT#0 TO UINT#87 DO
        IF (SecurityAccessFailureEncoder.Buffer[Index] <> ExpectedSecurityAccessFailure[Index]) AND (MismatchIndex = UINT#65535) THEN
            SecurityAccessFailurePassed := FALSE;
            MismatchIndex := Index;
        END_IF;
    END_FOR;
END_IF;

IF ParameterChangeRealPassed THEN
    FOR Index := UINT#0 TO UINT#111 DO
        IF (ParameterChangeRealEncoder.Buffer[Index] <> ExpectedParameterChangeReal[Index]) AND (MismatchIndex = UINT#65535) THEN
            ParameterChangeRealPassed := FALSE;
            MismatchIndex := Index;
        END_IF;
    END_FOR;
END_IF;

IF ParameterChangeIntPassed THEN
    FOR Index := UINT#0 TO UINT#103 DO
        IF (ParameterChangeIntEncoder.Buffer[Index] <> ExpectedParameterChangeInt[Index]) AND (MismatchIndex = UINT#65535) THEN
            ParameterChangeIntPassed := FALSE;
            MismatchIndex := Index;
        END_IF;
    END_FOR;
END_IF;

IF ParameterChangeBitsPassed THEN
    FOR Index := UINT#0 TO UINT#99 DO
        IF (ParameterChangeBitsEncoder.Buffer[Index] <> ExpectedParameterChangeBits[Index]) AND (MismatchIndex = UINT#65535) THEN
            ParameterChangeBitsPassed := FALSE;
            MismatchIndex := Index;
        END_IF;
    END_FOR;
END_IF;

IF ParameterChangeStringPassed THEN
    FOR Index := UINT#0 TO UINT#111 DO
        IF (ParameterChangeStringEncoder.Buffer[Index] <> ExpectedParameterChangeString[Index]) AND (MismatchIndex = UINT#65535) THEN
            ParameterChangeStringPassed := FALSE;
            MismatchIndex := Index;
        END_IF;
    END_FOR;
END_IF;

Passed := OperatorActionPassed AND OperatorLoginPassed AND OperatorLogoutPassed AND SecurityAccessFailurePassed AND ParameterChangeRealPassed AND ParameterChangeIntPassed AND ParameterChangeBitsPassed AND ParameterChangeStringPassed;
END_FUNCTION_BLOCK

(* ---- test_conformant_source_high_water.st ---- *)
FUNCTION_BLOCK OPENOT_TestConformantSourceHighWater
VAR_OUTPUT
    Passed : BOOL;
    MismatchIndex : UINT;
    ActualLength : UINT;
    ExpectedLength : UINT;
END_VAR
VAR
    Encoder : OPENOT_EncodeConformantSourceHighWater;
    Expected : ARRAY[0..55] OF BYTE := [
        BYTE#16#4F, BYTE#16#4F, BYTE#16#54, BYTE#16#32, BYTE#16#38, BYTE#16#00, BYTE#16#08, BYTE#16#00,
        BYTE#16#00, BYTE#16#00, BYTE#16#00, BYTE#16#00, BYTE#16#00, BYTE#16#00, BYTE#16#00, BYTE#16#00,
        BYTE#16#01, BYTE#16#00, BYTE#16#00, BYTE#16#00, BYTE#16#00, BYTE#16#00, BYTE#16#00, BYTE#16#00,
        BYTE#16#05, BYTE#16#00, BYTE#16#00, BYTE#16#00, BYTE#16#00, BYTE#16#00, BYTE#16#00, BYTE#16#00,
        BYTE#16#58, BYTE#16#00, BYTE#16#00, BYTE#16#00, BYTE#16#08, BYTE#16#01, BYTE#16#00, BYTE#16#80,
        BYTE#16#38, BYTE#16#00, BYTE#16#07, BYTE#16#08, BYTE#16#05, BYTE#16#00, BYTE#16#00, BYTE#16#00,
        BYTE#16#00, BYTE#16#00, BYTE#16#00, BYTE#16#00, BYTE#16#CD, BYTE#16#D4, BYTE#16#74, BYTE#16#86
    ];
    Index : UINT;
END_VAR

Encoder();
ActualLength := Encoder.Length;
ExpectedLength := UINT#56;
Passed := ActualLength = ExpectedLength;
MismatchIndex := UINT#65535;

IF Passed THEN
    FOR Index := UINT#0 TO ExpectedLength - UINT#1 DO
        IF (Encoder.Buffer[Index] <> Expected[Index]) AND (MismatchIndex = UINT#65535) THEN
            Passed := FALSE;
            MismatchIndex := Index;
        END_IF;
    END_FOR;
END_IF;
END_FUNCTION_BLOCK

(* ---- test_conformant_state_transition.st ---- *)
FUNCTION_BLOCK OPENOT_TestConformantStateTransition
VAR_OUTPUT
    Passed : BOOL;
    MismatchIndex : UINT;
    ActualLength : UINT;
    ExpectedLength : UINT;
END_VAR
VAR
    Encoder : OPENOT_EncodeConformantStateTransition;
    Expected : ARRAY[0..75] OF BYTE := [
        BYTE#16#4F, BYTE#16#4F, BYTE#16#54, BYTE#16#32, BYTE#16#4C, BYTE#16#00, BYTE#16#08, BYTE#16#00,
        BYTE#16#00, BYTE#16#CA, BYTE#16#9A, BYTE#16#3B, BYTE#16#00, BYTE#16#00, BYTE#16#00, BYTE#16#00,
        BYTE#16#01, BYTE#16#00, BYTE#16#00, BYTE#16#00, BYTE#16#00, BYTE#16#00, BYTE#16#00, BYTE#16#00,
        BYTE#16#01, BYTE#16#00, BYTE#16#00, BYTE#16#00, BYTE#16#00, BYTE#16#00, BYTE#16#00, BYTE#16#00,
        BYTE#16#42, BYTE#16#00, BYTE#16#00, BYTE#16#00, BYTE#16#01, BYTE#16#00, BYTE#16#00, BYTE#16#00,
        BYTE#16#01, BYTE#16#00, BYTE#16#05, BYTE#16#04, BYTE#16#07, BYTE#16#00, BYTE#16#00, BYTE#16#00,
        BYTE#16#02, BYTE#16#00, BYTE#16#03, BYTE#16#02, BYTE#16#02, BYTE#16#00, BYTE#16#00, BYTE#16#00,
        BYTE#16#03, BYTE#16#00, BYTE#16#03, BYTE#16#02, BYTE#16#03, BYTE#16#00, BYTE#16#00, BYTE#16#00,
        BYTE#16#04, BYTE#16#00, BYTE#16#03, BYTE#16#02, BYTE#16#04, BYTE#16#00, BYTE#16#00, BYTE#16#00,
        BYTE#16#60, BYTE#16#A3, BYTE#16#A5, BYTE#16#47
    ];
    Index : UINT;
END_VAR

Encoder();
ActualLength := Encoder.Length;
ExpectedLength := UINT#76;
Passed := ActualLength = ExpectedLength;
MismatchIndex := UINT#65535;

IF Passed THEN
    FOR Index := UINT#0 TO ExpectedLength - UINT#1 DO
        IF (Encoder.Buffer[Index] <> Expected[Index]) AND (MismatchIndex = UINT#65535) THEN
            Passed := FALSE;
            MismatchIndex := Index;
        END_IF;
    END_FOR;
END_IF;
END_FUNCTION_BLOCK

(* ---- test_conformant_value_changed_int.st ---- *)
FUNCTION_BLOCK OPENOT_TestConformantValueChangedInt
VAR_OUTPUT
    Passed : BOOL;
    MismatchIndex : UINT;
    ActualLength : UINT;
    ExpectedLength : UINT;
END_VAR
VAR
    Encoder : OPENOT_EncodeValueChangedInt;
    Expected : ARRAY[0..75] OF BYTE := [
        BYTE#16#4F, BYTE#16#4F, BYTE#16#54, BYTE#16#32, BYTE#16#4C, BYTE#16#00, BYTE#16#08, BYTE#16#00,
        BYTE#16#1E, BYTE#16#CA, BYTE#16#9A, BYTE#16#3B, BYTE#16#00, BYTE#16#00, BYTE#16#00, BYTE#16#00,
        BYTE#16#01, BYTE#16#00, BYTE#16#00, BYTE#16#00, BYTE#16#00, BYTE#16#00, BYTE#16#00, BYTE#16#00,
        BYTE#16#04, BYTE#16#00, BYTE#16#00, BYTE#16#00, BYTE#16#00, BYTE#16#00, BYTE#16#00, BYTE#16#00,
        BYTE#16#42, BYTE#16#00, BYTE#16#00, BYTE#16#00, BYTE#16#02, BYTE#16#00, BYTE#16#00, BYTE#16#00,
        BYTE#16#0D, BYTE#16#00, BYTE#16#05, BYTE#16#04, BYTE#16#D2, BYTE#16#07, BYTE#16#00, BYTE#16#00,
        BYTE#16#0F, BYTE#16#00, BYTE#16#06, BYTE#16#04, BYTE#16#28, BYTE#16#00, BYTE#16#00, BYTE#16#00,
        BYTE#16#10, BYTE#16#00, BYTE#16#06, BYTE#16#04, BYTE#16#2A, BYTE#16#00, BYTE#16#00, BYTE#16#00,
        BYTE#16#11, BYTE#16#00, BYTE#16#03, BYTE#16#02, BYTE#16#00, BYTE#16#00, BYTE#16#00, BYTE#16#00,
        BYTE#16#A1, BYTE#16#BB, BYTE#16#E9, BYTE#16#2E
    ];
    Index : UINT;
END_VAR

Encoder(
    SourceId := UDINT#66,
    RunId := ULINT#1,
    Seq := ULINT#4,
    SourceTime := ULINT#1000000030,
    ValueId := UDINT#2002,
    NewValue := DINT#42,
    HasPrevious := TRUE,
    PreviousValue := DINT#40,
    HasQuality := TRUE,
    Quality := UINT#0);
ActualLength := Encoder.Length;
ExpectedLength := UINT#76;
Passed := ActualLength = ExpectedLength;
MismatchIndex := UINT#65535;

IF Passed THEN
    FOR Index := UINT#0 TO ExpectedLength - UINT#1 DO
        IF (Encoder.Buffer[Index] <> Expected[Index]) AND (MismatchIndex = UINT#65535) THEN
            Passed := FALSE;
            MismatchIndex := Index;
        END_IF;
    END_FOR;
END_IF;
END_FUNCTION_BLOCK

(* ---- test_control_block.st ---- *)
FUNCTION_BLOCK OPENOT_TestControlBlock
VAR_OUTPUT
    Passed : BOOL;
    MismatchIndex : UINT;
    ActualLength : UINT;
    ExpectedLength : UINT;
END_VAR
VAR
    Writer : OPENOT_WriteControlBlockFixture;
    Expected : ARRAY[0..87] OF BYTE := [
        BYTE#16#4F, BYTE#16#4F, BYTE#16#54, BYTE#16#32, BYTE#16#02, BYTE#16#03, BYTE#16#00, BYTE#16#00,
        BYTE#16#07, BYTE#16#00, BYTE#16#00, BYTE#16#00, BYTE#16#00, BYTE#16#10, BYTE#16#00, BYTE#16#00,
        BYTE#16#02, BYTE#16#00, BYTE#16#00, BYTE#16#00, BYTE#16#00, BYTE#16#00, BYTE#16#00, BYTE#16#00,
        BYTE#16#00, BYTE#16#20, BYTE#16#00, BYTE#16#00, BYTE#16#00, BYTE#16#00, BYTE#16#00, BYTE#16#00,
        BYTE#16#00, BYTE#16#18, BYTE#16#00, BYTE#16#00, BYTE#16#00, BYTE#16#00, BYTE#16#00, BYTE#16#00,
        BYTE#16#0C, BYTE#16#00, BYTE#16#00, BYTE#16#00, BYTE#16#00, BYTE#16#00, BYTE#16#00, BYTE#16#00,
        BYTE#16#03, BYTE#16#00, BYTE#16#00, BYTE#16#00, BYTE#16#00, BYTE#16#00, BYTE#16#00, BYTE#16#00,
        BYTE#16#05, BYTE#16#00, BYTE#16#00, BYTE#16#00, BYTE#16#00, BYTE#16#00, BYTE#16#00, BYTE#16#00,
        BYTE#16#58, BYTE#16#1B, BYTE#16#00, BYTE#16#00, BYTE#16#00, BYTE#16#00, BYTE#16#00, BYTE#16#00,
        BYTE#16#64, BYTE#16#65, BYTE#16#66, BYTE#16#68, BYTE#16#61, BYTE#16#73, BYTE#16#68, BYTE#16#31,
        BYTE#16#6F, BYTE#16#6C, BYTE#16#64, BYTE#16#68, BYTE#16#61, BYTE#16#73, BYTE#16#68, BYTE#16#31
    ];
    Index : UINT;
END_VAR

Writer();
ActualLength := Writer.Length;
ExpectedLength := UINT#88;
Passed := ActualLength = ExpectedLength;
MismatchIndex := UINT#65535;

IF Passed THEN
    FOR Index := UINT#0 TO ExpectedLength - UINT#1 DO
        IF (Writer.Buffer[Index] <> Expected[Index]) AND (MismatchIndex = UINT#65535) THEN
            Passed := FALSE;
            MismatchIndex := Index;
        END_IF;
    END_FOR;
END_IF;
END_FUNCTION_BLOCK

(* ---- test_crc32c_kat.st ---- *)
FUNCTION_BLOCK OPENOT_TestCrc32cKat
VAR_OUTPUT
    Passed : BOOL;
    MismatchIndex : UINT;
    ActualLength : UINT;
    ExpectedLength : UINT;
    ActualCrc : DWORD;
    ExpectedCrc : DWORD;
END_VAR
VAR
    Data : OPENOT_BYTE_BUFFER;
END_VAR

Data[0] := BYTE#16#31;
Data[1] := BYTE#16#32;
Data[2] := BYTE#16#33;
Data[3] := BYTE#16#34;
Data[4] := BYTE#16#35;
Data[5] := BYTE#16#36;
Data[6] := BYTE#16#37;
Data[7] := BYTE#16#38;
Data[8] := BYTE#16#39;

ActualLength := UINT#9;
ExpectedLength := UINT#9;
ActualCrc := OPENOT_Crc32c(Data := Data, Length := UINT#9);
ExpectedCrc := DWORD#16#E3069283;
Passed := ActualCrc = ExpectedCrc;

IF Passed THEN
    MismatchIndex := UINT#65535;
ELSE
    MismatchIndex := UINT#0;
END_IF;
END_FUNCTION_BLOCK

(* ---- test_definition_changed.st ---- *)
FUNCTION_BLOCK OPENOT_TestDefinitionChanged
VAR_OUTPUT
    Passed : BOOL;
    MismatchIndex : UINT;
    ActualLength : UINT;
    ExpectedLength : UINT;
END_VAR
VAR
    Encoder : OPENOT_EncodeDefinitionChanged;
    DefHashOld : OPENOT_HASH8 := [
        BYTE#16#6F, BYTE#16#6C, BYTE#16#64, BYTE#16#68,
        BYTE#16#61, BYTE#16#73, BYTE#16#68, BYTE#16#31
    ];
    DefHashNew : OPENOT_HASH8 := [
        BYTE#16#6E, BYTE#16#65, BYTE#16#77, BYTE#16#68,
        BYTE#16#61, BYTE#16#73, BYTE#16#68, BYTE#16#32
    ];
    Expected : ARRAY[0..79] OF BYTE := [
        BYTE#16#4F, BYTE#16#4F, BYTE#16#54, BYTE#16#32, BYTE#16#50, BYTE#16#00, BYTE#16#08, BYTE#16#00,
        BYTE#16#00, BYTE#16#00, BYTE#16#00, BYTE#16#00, BYTE#16#00, BYTE#16#00, BYTE#16#00, BYTE#16#00,
        BYTE#16#01, BYTE#16#00, BYTE#16#00, BYTE#16#00, BYTE#16#00, BYTE#16#00, BYTE#16#00, BYTE#16#00,
        BYTE#16#01, BYTE#16#00, BYTE#16#00, BYTE#16#00, BYTE#16#00, BYTE#16#00, BYTE#16#00, BYTE#16#00,
        BYTE#16#00, BYTE#16#00, BYTE#16#00, BYTE#16#00, BYTE#16#06, BYTE#16#01, BYTE#16#00, BYTE#16#00,
        BYTE#16#39, BYTE#16#00, BYTE#16#0D, BYTE#16#08, BYTE#16#6F, BYTE#16#6C, BYTE#16#64, BYTE#16#68,
        BYTE#16#61, BYTE#16#73, BYTE#16#68, BYTE#16#31, BYTE#16#1C, BYTE#16#00, BYTE#16#0D, BYTE#16#08,
        BYTE#16#6E, BYTE#16#65, BYTE#16#77, BYTE#16#68, BYTE#16#61, BYTE#16#73, BYTE#16#68, BYTE#16#32,
        BYTE#16#3A, BYTE#16#00, BYTE#16#07, BYTE#16#08, BYTE#16#02, BYTE#16#00, BYTE#16#00, BYTE#16#00,
        BYTE#16#00, BYTE#16#00, BYTE#16#00, BYTE#16#00, BYTE#16#A5, BYTE#16#41, BYTE#16#2E, BYTE#16#B1
    ];
    Index : UINT;
END_VAR

Encoder(
    RunId := ULINT#1,
    Seq := ULINT#1,
    DefHashOld := DefHashOld,
    DefHashNew := DefHashNew,
    EpochId := ULINT#2,
    SourceTime := ULINT#0);
ActualLength := Encoder.Length;
ExpectedLength := UINT#80;
Passed := ActualLength = ExpectedLength;
MismatchIndex := UINT#65535;

IF Passed THEN
    FOR Index := UINT#0 TO ExpectedLength - UINT#1 DO
        IF (Encoder.Buffer[Index] <> Expected[Index]) AND (MismatchIndex = UINT#65535) THEN
            Passed := FALSE;
            MismatchIndex := Index;
        END_IF;
    END_FOR;
END_IF;
END_FUNCTION_BLOCK

(* ---- test_logger_started_cold.st ---- *)
FUNCTION_BLOCK OPENOT_TestLoggerStartedCold
VAR_OUTPUT
    Passed : BOOL;
    MismatchIndex : UINT;
    ActualLength : UINT;
    ExpectedLength : UINT;
END_VAR
VAR
    Encoder : OPENOT_EncodeLoggerStarted;
    Expected : ARRAY[0..51] OF BYTE := [
        BYTE#16#4F, BYTE#16#4F, BYTE#16#54, BYTE#16#32, BYTE#16#34, BYTE#16#00, BYTE#16#08, BYTE#16#00,
        BYTE#16#00, BYTE#16#00, BYTE#16#00, BYTE#16#00, BYTE#16#00, BYTE#16#00, BYTE#16#00, BYTE#16#00,
        BYTE#16#02, BYTE#16#00, BYTE#16#00, BYTE#16#00, BYTE#16#00, BYTE#16#00, BYTE#16#00, BYTE#16#00,
        BYTE#16#00, BYTE#16#00, BYTE#16#00, BYTE#16#00, BYTE#16#00, BYTE#16#00, BYTE#16#00, BYTE#16#00,
        BYTE#16#00, BYTE#16#00, BYTE#16#00, BYTE#16#00, BYTE#16#01, BYTE#16#01, BYTE#16#00, BYTE#16#00,
        BYTE#16#3B, BYTE#16#00, BYTE#16#00, BYTE#16#01, BYTE#16#01, BYTE#16#00, BYTE#16#00, BYTE#16#00,
        BYTE#16#CF, BYTE#16#2A, BYTE#16#DF, BYTE#16#09
    ];
    Index : UINT;
END_VAR

Encoder(RunId := ULINT#2, Seq := ULINT#0, ColdStart := TRUE, SourceTime := ULINT#0);
ActualLength := Encoder.Length;
ExpectedLength := UINT#52;
Passed := ActualLength = ExpectedLength;
MismatchIndex := UINT#65535;

IF Passed THEN
    FOR Index := UINT#0 TO ExpectedLength - UINT#1 DO
        IF (Encoder.Buffer[Index] <> Expected[Index]) AND (MismatchIndex = UINT#65535) THEN
            Passed := FALSE;
            MismatchIndex := Index;
        END_IF;
    END_FOR;
END_IF;
END_FUNCTION_BLOCK

(* ---- test_logger_started_warm.st ---- *)
FUNCTION_BLOCK OPENOT_TestLoggerStartedWarm
VAR_OUTPUT
    Passed : BOOL;
    MismatchIndex : UINT;
    ActualLength : UINT;
    ExpectedLength : UINT;
END_VAR
VAR
    Encoder : OPENOT_EncodeLoggerStarted;
    Expected : ARRAY[0..51] OF BYTE := [
        BYTE#16#4F, BYTE#16#4F, BYTE#16#54, BYTE#16#32, BYTE#16#34, BYTE#16#00, BYTE#16#08, BYTE#16#00,
        BYTE#16#00, BYTE#16#00, BYTE#16#00, BYTE#16#00, BYTE#16#00, BYTE#16#00, BYTE#16#00, BYTE#16#00,
        BYTE#16#01, BYTE#16#00, BYTE#16#00, BYTE#16#00, BYTE#16#00, BYTE#16#00, BYTE#16#00, BYTE#16#00,
        BYTE#16#02, BYTE#16#00, BYTE#16#00, BYTE#16#00, BYTE#16#00, BYTE#16#00, BYTE#16#00, BYTE#16#00,
        BYTE#16#00, BYTE#16#00, BYTE#16#00, BYTE#16#00, BYTE#16#01, BYTE#16#01, BYTE#16#00, BYTE#16#00,
        BYTE#16#3B, BYTE#16#00, BYTE#16#00, BYTE#16#01, BYTE#16#00, BYTE#16#00, BYTE#16#00, BYTE#16#00,
        BYTE#16#C7, BYTE#16#02, BYTE#16#02, BYTE#16#E3
    ];
    Index : UINT;
END_VAR

Encoder(RunId := ULINT#1, Seq := ULINT#2, ColdStart := FALSE, SourceTime := ULINT#0);
ActualLength := Encoder.Length;
ExpectedLength := UINT#52;
Passed := ActualLength = ExpectedLength;
MismatchIndex := UINT#65535;

IF Passed THEN
    FOR Index := UINT#0 TO ExpectedLength - UINT#1 DO
        IF (Encoder.Buffer[Index] <> Expected[Index]) AND (MismatchIndex = UINT#65535) THEN
            Passed := FALSE;
            MismatchIndex := Index;
        END_IF;
    END_FOR;
END_IF;
END_FUNCTION_BLOCK

(* ---- test_logger_stopped.st ---- *)
FUNCTION_BLOCK OPENOT_TestLoggerStopped
VAR_OUTPUT
    Passed : BOOL;
    MismatchIndex : UINT;
    ActualLength : UINT;
    ExpectedLength : UINT;
END_VAR
VAR
    Encoder : OPENOT_EncodeLoggerStopped;
    Expected : ARRAY[0..43] OF BYTE := [
        BYTE#16#4F, BYTE#16#4F, BYTE#16#54, BYTE#16#32, BYTE#16#2C, BYTE#16#00, BYTE#16#08, BYTE#16#00,
        BYTE#16#00, BYTE#16#00, BYTE#16#00, BYTE#16#00, BYTE#16#00, BYTE#16#00, BYTE#16#00, BYTE#16#00,
        BYTE#16#01, BYTE#16#00, BYTE#16#00, BYTE#16#00, BYTE#16#00, BYTE#16#00, BYTE#16#00, BYTE#16#00,
        BYTE#16#00, BYTE#16#00, BYTE#16#00, BYTE#16#00, BYTE#16#00, BYTE#16#00, BYTE#16#00, BYTE#16#00,
        BYTE#16#00, BYTE#16#00, BYTE#16#00, BYTE#16#00, BYTE#16#02, BYTE#16#01, BYTE#16#00, BYTE#16#00,
        BYTE#16#09, BYTE#16#A8, BYTE#16#70, BYTE#16#85
    ];
    Index : UINT;
END_VAR

Encoder(RunId := ULINT#1, Seq := ULINT#0, SourceTime := ULINT#0);
ActualLength := Encoder.Length;
ExpectedLength := UINT#44;
Passed := ActualLength = ExpectedLength;
MismatchIndex := UINT#65535;

IF Passed THEN
    FOR Index := UINT#0 TO ExpectedLength - UINT#1 DO
        IF (Encoder.Buffer[Index] <> Expected[Index]) AND (MismatchIndex = UINT#65535) THEN
            Passed := FALSE;
            MismatchIndex := Index;
        END_IF;
    END_FOR;
END_IF;
END_FUNCTION_BLOCK

(* ---- test_loss_range_formation.st ---- *)
FUNCTION_BLOCK OPENOT_EncodeFormationMinimalMessage
VAR_INPUT
    SourceId : UDINT;
    Seq : ULINT;
END_VAR
VAR_OUTPUT
    Buffer : OPENOT_BYTE_BUFFER;
    Length : UINT;
END_VAR
VAR
    Pos : UINT;
    Crc : DWORD;
END_VAR

Pos := OPENOT_WriteHeader(
    TotalLength := UINT#44,
    Flags := UINT#16#0008,
    SourceTime := ULINT#1780000000000000000 + Seq,
    RunId := ULINT#1,
    Seq := Seq,
    SourceId := SourceId,
    EventTypeId := UDINT#16#0003,
    Buffer := Buffer);

Crc := OPENOT_Crc32c(Data := Buffer, Length := Pos);
Pos := OPENOT_WriteDWordLE(Offset := Pos, Value := Crc, Buffer := Buffer);
Length := Pos;
END_FUNCTION_BLOCK

FUNCTION_BLOCK OPENOT_TestLossRangeFormation
VAR_OUTPUT
    Passed : BOOL;
    FoundSource : BOOL;
    ActualFirstSeq : ULINT;
    ActualLastSeq : ULINT;
    ActualCount : ULINT;
    ActualLossRangeCount : UINT;
    ActualLostCount : ULINT;
END_VAR
VAR
    Producer : OPENOT_Ring256Producer;
    Encoder : OPENOT_EncodeFormationMinimalMessage;
    SeqIndex : UINT;
    LossIndex : UINT;
    SeqValue : ULINT;
    Ran : BOOL;
END_VAR

IF NOT Ran THEN
    FOR SeqIndex := UINT#0 TO UINT#4 DO
        SeqValue := UINT_TO_ULINT(SeqIndex);
        Encoder(SourceId := UDINT#88, Seq := SeqValue);
        Producer(
            Execute := TRUE,
            Record := Encoder.Buffer,
            Length := Encoder.Length,
            RunId := ULINT#1,
            SourceId := UDINT#88,
            Seq := SeqValue);
    END_FOR;

    FOR SeqIndex := UINT#0 TO UINT#79 DO
        SeqValue := UINT_TO_ULINT(SeqIndex);
        Encoder(SourceId := UDINT#99, Seq := SeqValue);
        Producer(
            Execute := TRUE,
            Record := Encoder.Buffer,
            Length := Encoder.Length,
            RunId := ULINT#1,
            SourceId := UDINT#99,
            Seq := SeqValue);
    END_FOR;

    Ran := TRUE;
END_IF;

FoundSource := FALSE;
ActualFirstSeq := ULINT#0;
ActualLastSeq := ULINT#0;
ActualCount := ULINT#0;
ActualLossRangeCount := Producer.LossRangeCount;
ActualLostCount := Producer.LostCount;

IF Producer.LossRangeCount > UINT#0 THEN
    FOR LossIndex := UINT#0 TO Producer.LossRangeCount - UINT#1 DO
        IF (Producer.LossRanges[LossIndex].RunId = ULINT#1) AND (Producer.LossRanges[LossIndex].SourceId = UDINT#88) AND (NOT FoundSource) THEN
            FoundSource := TRUE;
            ActualFirstSeq := Producer.LossRanges[LossIndex].FirstSeq;
            ActualLastSeq := Producer.LossRanges[LossIndex].LastSeq;
            ActualCount := (ActualLastSeq - ActualFirstSeq) + ULINT#1;
        END_IF;
    END_FOR;
END_IF;

Passed :=
    FoundSource AND
    (ActualFirstSeq = ULINT#0) AND
    (ActualLastSeq = ULINT#4) AND
    (ActualCount = ULINT#5) AND
    (NOT Producer.LossRangeOverflow) AND
    (NOT Producer.Error);
END_FUNCTION_BLOCK

(* ---- test_loss_range_interleaved.st ---- *)
FUNCTION_BLOCK OPENOT_EncodeInterleavedMinimalMessage
VAR_INPUT
    SourceId : UDINT;
    Seq : ULINT;
END_VAR
VAR_OUTPUT
    Buffer : OPENOT_BYTE_BUFFER;
    Length : UINT;
END_VAR
VAR
    Pos : UINT;
    Crc : DWORD;
END_VAR

Pos := OPENOT_WriteHeader(
    TotalLength := UINT#44,
    Flags := UINT#16#0008,
    SourceTime := ULINT#1780000000000000000 + Seq,
    RunId := ULINT#1,
    Seq := Seq,
    SourceId := SourceId,
    EventTypeId := UDINT#16#0003,
    Buffer := Buffer);

Crc := OPENOT_Crc32c(Data := Buffer, Length := Pos);
Pos := OPENOT_WriteDWordLE(Offset := Pos, Value := Crc, Buffer := Buffer);
Length := Pos;
END_FUNCTION_BLOCK

FUNCTION_BLOCK OPENOT_TestLossRangeInterleaved
VAR_OUTPUT
    Passed : BOOL;
    ActualLossRangeCount : UINT;
    ActualLostCount : ULINT;
END_VAR
VAR
    Producer : OPENOT_Ring256Producer;
    Encoder : OPENOT_EncodeInterleavedMinimalMessage;
    Ran : BOOL;
END_VAR

IF NOT Ran THEN
    Encoder(SourceId := UDINT#10, Seq := ULINT#0);
    Producer(
        Execute := TRUE,
        Record := Encoder.Buffer,
        Length := Encoder.Length,
        RunId := ULINT#1,
        SourceId := UDINT#10,
        Seq := ULINT#0);
    Encoder(SourceId := UDINT#20, Seq := ULINT#0);
    Producer(
        Execute := TRUE,
        Record := Encoder.Buffer,
        Length := Encoder.Length,
        RunId := ULINT#1,
        SourceId := UDINT#20,
        Seq := ULINT#0);
    Encoder(SourceId := UDINT#10, Seq := ULINT#1);
    Producer(
        Execute := TRUE,
        Record := Encoder.Buffer,
        Length := Encoder.Length,
        RunId := ULINT#1,
        SourceId := UDINT#10,
        Seq := ULINT#1);
    Encoder(SourceId := UDINT#20, Seq := ULINT#1);
    Producer(
        Execute := TRUE,
        Record := Encoder.Buffer,
        Length := Encoder.Length,
        RunId := ULINT#1,
        SourceId := UDINT#20,
        Seq := ULINT#1);
    Encoder(SourceId := UDINT#10, Seq := ULINT#2);
    Producer(
        Execute := TRUE,
        Record := Encoder.Buffer,
        Length := Encoder.Length,
        RunId := ULINT#1,
        SourceId := UDINT#10,
        Seq := ULINT#2);
    Encoder(SourceId := UDINT#20, Seq := ULINT#2);
    Producer(
        Execute := TRUE,
        Record := Encoder.Buffer,
        Length := Encoder.Length,
        RunId := ULINT#1,
        SourceId := UDINT#20,
        Seq := ULINT#2);
    Encoder(SourceId := UDINT#10, Seq := ULINT#3);
    Producer(
        Execute := TRUE,
        Record := Encoder.Buffer,
        Length := Encoder.Length,
        RunId := ULINT#1,
        SourceId := UDINT#10,
        Seq := ULINT#3);
    Encoder(SourceId := UDINT#20, Seq := ULINT#3);
    Producer(
        Execute := TRUE,
        Record := Encoder.Buffer,
        Length := Encoder.Length,
        RunId := ULINT#1,
        SourceId := UDINT#20,
        Seq := ULINT#3);
    Encoder(SourceId := UDINT#10, Seq := ULINT#4);
    Producer(
        Execute := TRUE,
        Record := Encoder.Buffer,
        Length := Encoder.Length,
        RunId := ULINT#1,
        SourceId := UDINT#10,
        Seq := ULINT#4);

    Ran := TRUE;
END_IF;

ActualLossRangeCount := Producer.LossRangeCount;
ActualLostCount := Producer.LostCount;

Passed :=
    (Producer.LossRangeCount = UINT#4) AND
    (Producer.LostCount = ULINT#4) AND
    (Producer.LossRanges[0].RunId = ULINT#1) AND
    (Producer.LossRanges[0].SourceId = UDINT#10) AND
    (Producer.LossRanges[0].FirstSeq = ULINT#0) AND
    (Producer.LossRanges[0].LastSeq = ULINT#0) AND
    (Producer.LossRanges[1].RunId = ULINT#1) AND
    (Producer.LossRanges[1].SourceId = UDINT#20) AND
    (Producer.LossRanges[1].FirstSeq = ULINT#0) AND
    (Producer.LossRanges[1].LastSeq = ULINT#0) AND
    (Producer.LossRanges[2].RunId = ULINT#1) AND
    (Producer.LossRanges[2].SourceId = UDINT#10) AND
    (Producer.LossRanges[2].FirstSeq = ULINT#1) AND
    (Producer.LossRanges[2].LastSeq = ULINT#1) AND
    (Producer.LossRanges[3].RunId = ULINT#1) AND
    (Producer.LossRanges[3].SourceId = UDINT#20) AND
    (Producer.LossRanges[3].FirstSeq = ULINT#1) AND
    (Producer.LossRanges[3].LastSeq = ULINT#1) AND
    (NOT Producer.LossRangeOverflow) AND
    (NOT Producer.Error);
END_FUNCTION_BLOCK

(* ---- test_minimal_message.st ---- *)
FUNCTION_BLOCK OPENOT_TestMinimalMessage
VAR_OUTPUT
    Passed : BOOL;
    MismatchIndex : UINT;
    ActualLength : UINT;
    ExpectedLength : UINT;
END_VAR
VAR
    Encoder : OPENOT_EncodeMinimalMessage;
    Expected : ARRAY[0..43] OF BYTE := [
        BYTE#16#4F, BYTE#16#4F, BYTE#16#54, BYTE#16#32, BYTE#16#2C, BYTE#16#00, BYTE#16#08, BYTE#16#00,
        BYTE#16#03, BYTE#16#00, BYTE#16#32, BYTE#16#B4, BYTE#16#91, BYTE#16#D4, BYTE#16#B3, BYTE#16#18,
        BYTE#16#01, BYTE#16#00, BYTE#16#00, BYTE#16#00, BYTE#16#00, BYTE#16#00, BYTE#16#00, BYTE#16#00,
        BYTE#16#03, BYTE#16#00, BYTE#16#00, BYTE#16#00, BYTE#16#00, BYTE#16#00, BYTE#16#00, BYTE#16#00,
        BYTE#16#07, BYTE#16#00, BYTE#16#00, BYTE#16#00, BYTE#16#03, BYTE#16#00, BYTE#16#00, BYTE#16#00,
        BYTE#16#21, BYTE#16#52, BYTE#16#EF, BYTE#16#97
    ];
    Index : UINT;
END_VAR

Encoder(SourceId := UDINT#7, Seq := ULINT#3);
ActualLength := Encoder.Length;
ExpectedLength := UINT#44;
Passed := ActualLength = ExpectedLength;
MismatchIndex := UINT#65535;

IF Passed THEN
    FOR Index := UINT#0 TO ExpectedLength - UINT#1 DO
        IF (Encoder.Buffer[Index] <> Expected[Index]) AND (MismatchIndex = UINT#65535) THEN
            Passed := FALSE;
            MismatchIndex := Index;
        END_IF;
    END_FOR;
END_IF;
END_FUNCTION_BLOCK

(* ---- test_producer_checkpoint.st ---- *)
FUNCTION_BLOCK OPENOT_TestProducerCheckpoint
VAR_OUTPUT
    Passed : BOOL;
    ProducedCount : ULINT;
    NextSeqAfterCheckpoint : ULINT;
    EnvelopeSeqIsFive : BOOL;
    PayloadProducedCountIsFive : BOOL;
    CheckpointLength : UINT;
    CheckpointStartAbs : ULINT;
END_VAR
VAR
    Producer : OPENOT_Producer;
    Ran : BOOL;
    WritesOk : BOOL;
    SourceFound : BOOL;
    Index : UINT;
END_VAR

IF NOT Ran THEN
    WritesOk := TRUE;

    Producer(Execute := TRUE, SourceId := UDINT#88, Checkpoint := FALSE);
    WritesOk := WritesOk AND Producer.Done AND (NOT Producer.Error) AND (Producer.AssignedSeq = ULINT#0);
    Producer(Execute := TRUE, SourceId := UDINT#88, Checkpoint := FALSE);
    WritesOk := WritesOk AND Producer.Done AND (NOT Producer.Error) AND (Producer.AssignedSeq = ULINT#1);
    Producer(Execute := TRUE, SourceId := UDINT#88, Checkpoint := FALSE);
    WritesOk := WritesOk AND Producer.Done AND (NOT Producer.Error) AND (Producer.AssignedSeq = ULINT#2);
    Producer(Execute := TRUE, SourceId := UDINT#88, Checkpoint := FALSE);
    WritesOk := WritesOk AND Producer.Done AND (NOT Producer.Error) AND (Producer.AssignedSeq = ULINT#3);
    Producer(Execute := TRUE, SourceId := UDINT#88, Checkpoint := FALSE);
    WritesOk := WritesOk AND Producer.Done AND (NOT Producer.Error) AND (Producer.AssignedSeq = ULINT#4);

    Producer(Execute := TRUE, SourceId := UDINT#88, Checkpoint := TRUE);
    ProducedCount := Producer.ProducedCount;
    CheckpointLength := UINT#56;
    CheckpointStartAbs := Producer.LastStartAbs;

    EnvelopeSeqIsFive :=
        (Producer.Ring[24] = BYTE#16#05) AND
        (Producer.Ring[25] = BYTE#16#00) AND
        (Producer.Ring[26] = BYTE#16#00) AND
        (Producer.Ring[27] = BYTE#16#00) AND
        (Producer.Ring[28] = BYTE#16#00) AND
        (Producer.Ring[29] = BYTE#16#00) AND
        (Producer.Ring[30] = BYTE#16#00) AND
        (Producer.Ring[31] = BYTE#16#00);

    PayloadProducedCountIsFive :=
        (Producer.Ring[44] = BYTE#16#05) AND
        (Producer.Ring[45] = BYTE#16#00) AND
        (Producer.Ring[46] = BYTE#16#00) AND
        (Producer.Ring[47] = BYTE#16#00) AND
        (Producer.Ring[48] = BYTE#16#00) AND
        (Producer.Ring[49] = BYTE#16#00) AND
        (Producer.Ring[50] = BYTE#16#00) AND
        (Producer.Ring[51] = BYTE#16#00);

    Ran := TRUE;
END_IF;

SourceFound := FALSE;
NextSeqAfterCheckpoint := ULINT#0;
FOR Index := UINT#0 TO UINT#15 DO
    IF Producer.SourceUsed[Index] AND (Producer.SourceIds[Index] = UDINT#88) THEN
        SourceFound := TRUE;
        NextSeqAfterCheckpoint := Producer.SourceNextSeqs[Index];
    END_IF;
END_FOR;

Passed :=
    WritesOk AND
    Producer.Done AND
    Producer.CheckpointDone AND
    (NOT Producer.Error) AND
    (ProducedCount = ULINT#5) AND
    (CheckpointStartAbs = ULINT#256) AND
    (Producer.LastEndAbs = ULINT#312) AND
    (CheckpointLength = UINT#56) AND
    EnvelopeSeqIsFive AND
    PayloadProducedCountIsFive AND
    SourceFound AND
    (NextSeqAfterCheckpoint = ULINT#6);
END_FUNCTION_BLOCK

(* ---- test_producer_seq.st ---- *)
FUNCTION_BLOCK OPENOT_TestProducerSeq
VAR_OUTPUT
    Passed : BOOL;
    ASeq0 : ULINT;
    ASeq1 : ULINT;
    ASeq2 : ULINT;
    BSeq0 : ULINT;
    BSeq1 : ULINT;
    ANextSeq : ULINT;
    BNextSeq : ULINT;
    ReservedSourceRejected : BOOL;
    SourceTableFullRejected : BOOL;
    SourceCountAfterFill : UINT;
END_VAR
VAR
    Producer : OPENOT_Producer;
    ReservedProducer : OPENOT_Producer;
    FullProducer : OPENOT_Producer;
    Ran : BOOL;
    WritesOk : BOOL;
    FillOk : BOOL;
    AFound : BOOL;
    BFound : BOOL;
    Index : UINT;
    FillSource : UDINT;
END_VAR

IF NOT Ran THEN
    WritesOk := TRUE;
    FillOk := TRUE;

    Producer(Execute := TRUE, SourceId := UDINT#10);
    ASeq0 := Producer.AssignedSeq;
    WritesOk := WritesOk AND Producer.Done AND (NOT Producer.Error);
    Producer(Execute := FALSE, SourceId := UDINT#10);

    Producer(Execute := TRUE, SourceId := UDINT#10);
    ASeq1 := Producer.AssignedSeq;
    WritesOk := WritesOk AND Producer.Done AND (NOT Producer.Error);
    Producer(Execute := FALSE, SourceId := UDINT#10);

    Producer(Execute := TRUE, SourceId := UDINT#10);
    ASeq2 := Producer.AssignedSeq;
    WritesOk := WritesOk AND Producer.Done AND (NOT Producer.Error);
    Producer(Execute := FALSE, SourceId := UDINT#10);

    Producer(Execute := TRUE, SourceId := UDINT#20);
    BSeq0 := Producer.AssignedSeq;
    WritesOk := WritesOk AND Producer.Done AND (NOT Producer.Error);
    Producer(Execute := FALSE, SourceId := UDINT#20);

    Producer(Execute := TRUE, SourceId := UDINT#20);
    BSeq1 := Producer.AssignedSeq;
    WritesOk := WritesOk AND Producer.Done AND (NOT Producer.Error);
    Producer(Execute := FALSE, SourceId := UDINT#20);

    ReservedProducer(Execute := TRUE, SourceId := UDINT#0);
    ReservedSourceRejected := ReservedProducer.Error AND (NOT ReservedProducer.Done);
    ReservedProducer(Execute := FALSE, SourceId := UDINT#0);

    FOR Index := UINT#0 TO UINT#15 DO
        FillSource := UINT_TO_UDINT(Index) + UDINT#1;
        FullProducer(Execute := TRUE, SourceId := FillSource);
        FillOk :=
            FillOk AND
            FullProducer.Done AND
            (NOT FullProducer.Error) AND
            (NOT FullProducer.SourceTableFull);
        FullProducer(Execute := FALSE, SourceId := FillSource);
    END_FOR;

    SourceCountAfterFill := FullProducer.SourceCount;
    FullProducer(Execute := TRUE, SourceId := UDINT#17);
    SourceTableFullRejected :=
        FullProducer.Error AND
        FullProducer.SourceTableFull AND
        (NOT FullProducer.Done);

    Ran := TRUE;
END_IF;

AFound := FALSE;
BFound := FALSE;
ANextSeq := ULINT#0;
BNextSeq := ULINT#0;
FOR Index := UINT#0 TO UINT#15 DO
    IF Producer.SourceUsed[Index] AND (Producer.SourceIds[Index] = UDINT#10) THEN
        ANextSeq := Producer.SourceNextSeqs[Index];
        AFound := TRUE;
    END_IF;
    IF Producer.SourceUsed[Index] AND (Producer.SourceIds[Index] = UDINT#20) THEN
        BNextSeq := Producer.SourceNextSeqs[Index];
        BFound := TRUE;
    END_IF;
END_FOR;

Passed :=
    WritesOk AND
    (ASeq0 = ULINT#0) AND
    (ASeq1 = ULINT#1) AND
    (ASeq2 = ULINT#2) AND
    (BSeq0 = ULINT#0) AND
    (BSeq1 = ULINT#1) AND
    AFound AND
    BFound AND
    (ANextSeq = ULINT#3) AND
    (BNextSeq = ULINT#2) AND
    (Producer.SourceCount = UINT#2) AND
    ReservedSourceRejected AND
    FillOk AND
    (SourceCountAfterFill = UINT#16) AND
    SourceTableFullRejected;
END_FUNCTION_BLOCK

(* ---- test_published_record_count_durable.st ---- *)
FUNCTION_BLOCK OPENOT_TestPublishedRecordCountDurable
VAR_OUTPUT
    Passed : BOOL;
    PublishedRecordCount : ULINT;
    EmissionCount : UINT;
    FinalAssignedSeq : ULINT;
END_VAR
VAR
    Producer : OPENOT_Producer;
    Ran : BOOL;
    WritesOk : BOOL;
    Index : UINT;
    ExpectedSeq : ULINT;
END_VAR

IF NOT Ran THEN
    WritesOk := TRUE;
    ExpectedSeq := ULINT#0;

    FOR Index := UINT#0 TO UINT#39 DO
        Producer(Execute := TRUE, Op := UINT#0, SourceId := UDINT#77);
        FinalAssignedSeq := Producer.AssignedSeq;
        WritesOk :=
            WritesOk AND
            Producer.Done AND
            (NOT Producer.Error) AND
            (Producer.AssignedSeq = ExpectedSeq);
        Producer(Execute := FALSE, Op := UINT#0, SourceId := UDINT#77);
        ExpectedSeq := ExpectedSeq + ULINT#1;
    END_FOR;

    PublishedRecordCount := Producer.PublishedRecordCount;
    EmissionCount := Producer.EmissionCount;
    Ran := TRUE;
END_IF;

Passed :=
    WritesOk AND
    (PublishedRecordCount = ULINT#40) AND
    (EmissionCount = UINT#32) AND
    (FinalAssignedSeq = ULINT#39) AND
    (Producer.PublishedRecordCount = ULINT#40) AND
    (Producer.EmissionCount = UINT#32) AND
    (Producer.SourceCount = UINT#1);
END_FUNCTION_BLOCK

(* ---- test_records_dropped.st ---- *)
FUNCTION_BLOCK OPENOT_TestProducerRecordsDropped
VAR_OUTPUT
    Passed : BOOL;
    MismatchIndex : UINT;
    ActualLength : UINT;
    ExpectedLength : UINT;
END_VAR
VAR
    Encoder : OPENOT_EncodeProducerRecordsDropped;
    BadBounds : OPENOT_EncodeProducerRecordsDropped;
    BadCount : OPENOT_EncodeProducerRecordsDropped;
    Expected : ARRAY[0..75] OF BYTE := [
        (* EXPECTED_RECORDS_DROPPED_BEGIN *)
        BYTE#16#4F, BYTE#16#4F, BYTE#16#54, BYTE#16#32, BYTE#16#4C, BYTE#16#00, BYTE#16#08, BYTE#16#00,
        BYTE#16#00, BYTE#16#00, BYTE#16#00, BYTE#16#00, BYTE#16#00, BYTE#16#00, BYTE#16#00, BYTE#16#00,
        BYTE#16#09, BYTE#16#00, BYTE#16#00, BYTE#16#00, BYTE#16#00, BYTE#16#00, BYTE#16#00, BYTE#16#00,
        BYTE#16#2C, BYTE#16#00, BYTE#16#00, BYTE#16#00, BYTE#16#00, BYTE#16#00, BYTE#16#00, BYTE#16#00,
        BYTE#16#2A, BYTE#16#00, BYTE#16#00, BYTE#16#00, BYTE#16#04, BYTE#16#01, BYTE#16#00, BYTE#16#00,
        BYTE#16#16, BYTE#16#00, BYTE#16#05, BYTE#16#04, BYTE#16#05, BYTE#16#00, BYTE#16#00, BYTE#16#00,
        BYTE#16#17, BYTE#16#00, BYTE#16#07, BYTE#16#08, BYTE#16#64, BYTE#16#00, BYTE#16#00, BYTE#16#00,
        BYTE#16#00, BYTE#16#00, BYTE#16#00, BYTE#16#00, BYTE#16#18, BYTE#16#00, BYTE#16#07, BYTE#16#08,
        BYTE#16#68, BYTE#16#00, BYTE#16#00, BYTE#16#00, BYTE#16#00, BYTE#16#00, BYTE#16#00, BYTE#16#00,
        BYTE#16#57, BYTE#16#48, BYTE#16#CC, BYTE#16#E3
        (* EXPECTED_RECORDS_DROPPED_END *)
    ];
    Index : UINT;
END_VAR

Encoder(
    RunId := ULINT#9,
    SourceId := UDINT#42,
    FirstSeq := ULINT#100,
    LastSeq := ULINT#104,
    Seq := ULINT#44,
    SourceTime := ULINT#0);
BadBounds(
    RunId := ULINT#9,
    SourceId := UDINT#42,
    FirstSeq := ULINT#5,
    LastSeq := ULINT#4,
    Seq := ULINT#44,
    SourceTime := ULINT#0);
BadCount(
    RunId := ULINT#9,
    SourceId := UDINT#42,
    FirstSeq := ULINT#0,
    LastSeq := ULINT#4294967295,
    Seq := ULINT#44,
    SourceTime := ULINT#0);

ActualLength := Encoder.Length;
ExpectedLength := UINT#76;
Passed :=
    Encoder.Done AND
    (NOT Encoder.Error) AND
    BadBounds.Error AND
    (NOT BadBounds.Done) AND
    (BadBounds.Length = UINT#0) AND
    BadCount.Error AND
    (NOT BadCount.Done) AND
    (BadCount.Length = UINT#0) AND
    (ActualLength = ExpectedLength);
MismatchIndex := UINT#65535;

IF Passed THEN
    FOR Index := UINT#0 TO ExpectedLength - UINT#1 DO
        IF (Encoder.Buffer[Index] <> Expected[Index]) AND (MismatchIndex = UINT#65535) THEN
            Passed := FALSE;
            MismatchIndex := Index;
        END_IF;
    END_FOR;
END_IF;
END_FUNCTION_BLOCK

(* ---- test_scan_records_burst.st ---- *)
FUNCTION OPENOT_TestScanRecordCrcValid : BOOL
VAR_INPUT
    Records : OPENOT_SCAN_RECORD_BUFFER;
    Offset : UINT;
    Length : UINT;
END_VAR
VAR
    Work : OPENOT_BYTE_BUFFER;
    Index : UINT;
    CrcLength : UINT;
    ActualCrc : DWORD;
    ExpectedCrc : DWORD;
END_VAR

IF (Length < UINT#44) OR (Length > UINT#256) THEN
    OPENOT_TestScanRecordCrcValid := FALSE;
ELSE
    FOR Index := UINT#0 TO Length - UINT#1 DO
        Work[Index] := Records[Offset + Index];
    END_FOR;

    CrcLength := Length - UINT#4;
    ActualCrc := OPENOT_Crc32c(Data := Work, Length := CrcLength);
    ExpectedCrc :=
        BYTE_TO_DWORD(Work[Length - UINT#4]) OR
        SHL(BYTE_TO_DWORD(Work[Length - UINT#3]), UINT#8) OR
        SHL(BYTE_TO_DWORD(Work[Length - UINT#2]), UINT#16) OR
        SHL(BYTE_TO_DWORD(Work[Length - UINT#1]), UINT#24);
    OPENOT_TestScanRecordCrcValid := ActualCrc = ExpectedCrc;
END_IF;
END_FUNCTION

FUNCTION OPENOT_TestScanRecordHeaderOk : BOOL
VAR_INPUT
    Records : OPENOT_SCAN_RECORD_BUFFER;
    Offset : UINT;
    Length : UINT;
    EventTypeId : UDINT;
    SourceId : UDINT;
END_VAR
VAR
    HeaderOk : BOOL;
    SourceRemaining : UDINT;
    EventRemaining : UDINT;
    Index : UINT;
    Pos : UINT;
END_VAR

HeaderOk :=
    (Length >= UINT#44) AND
    (Records[Offset] = BYTE#16#4F) AND
    (Records[Offset + UINT#1] = BYTE#16#4F) AND
    (Records[Offset + UINT#2] = BYTE#16#54) AND
    (Records[Offset + UINT#3] = BYTE#16#32) AND
    (Records[Offset + UINT#4] = UINT_TO_BYTE(Length MOD UINT#256)) AND
    (Records[Offset + UINT#5] = UINT_TO_BYTE((Length / UINT#256) MOD UINT#256)) AND
    (Records[Offset + UINT#6] = BYTE#16#08) AND
    (Records[Offset + UINT#7] = BYTE#16#00);

SourceRemaining := SourceId;
FOR Index := UINT#0 TO UINT#3 DO
    Pos := Offset + UINT#32 + Index;
    HeaderOk := HeaderOk AND (Records[Pos] = UDINT_TO_BYTE(SourceRemaining MOD UDINT#256));
    SourceRemaining := SourceRemaining / UDINT#256;
END_FOR;

EventRemaining := EventTypeId;
FOR Index := UINT#0 TO UINT#3 DO
    Pos := Offset + UINT#36 + Index;
    HeaderOk := HeaderOk AND (Records[Pos] = UDINT_TO_BYTE(EventRemaining MOD UDINT#256));
    EventRemaining := EventRemaining / UDINT#256;
END_FOR;

OPENOT_TestScanRecordHeaderOk := HeaderOk;
END_FUNCTION

FUNCTION_BLOCK OPENOT_TestScanRecordsBurst
VAR_OUTPUT
    Passed : BOOL;
    SingleRecordOpsOk : BOOL;
    BurstCrcOk : BOOL;
    BurstOrderOk : BOOL;
    BurstContiguousOk : BOOL;
    BurstScanRecordCount : UINT;
    BurstPublishedDelta : ULINT;
    BurstBytes : UINT;
    DataScanRecordCount : UINT;
    DefinitionChangedScanRecordCount : UINT;
    LoggerStartedScanRecordCount : UINT;
    CheckpointScanRecordCount : UINT;
    BurstNoEdgeScanRecordCount : UINT;
    SingleNoEdgeScanRecordCount : UINT;
END_VAR
VAR
    Producer : OPENOT_Producer;
    DefHashOld : OPENOT_HASH8 := [
        BYTE#16#6F, BYTE#16#6C, BYTE#16#64, BYTE#16#68,
        BYTE#16#61, BYTE#16#73, BYTE#16#68, BYTE#16#31
    ];
    DefHashNew : OPENOT_HASH8 := [
        BYTE#16#6E, BYTE#16#65, BYTE#16#77, BYTE#16#68,
        BYTE#16#61, BYTE#16#73, BYTE#16#68, BYTE#16#32
    ];
    Ran : BOOL;
    OpsOk : BOOL;
    CountBefore : ULINT;
    Delta : ULINT;
    Offset0 : UINT;
    Offset1 : UINT;
    Offset2 : UINT;
    Length0 : UINT;
    Length1 : UINT;
    Length2 : UINT;
END_VAR

IF NOT Ran THEN
    OpsOk := TRUE;
    SingleRecordOpsOk := TRUE;

    Producer(Execute := TRUE, Op := UINT#0, SourceId := UDINT#30);
    CountBefore := ULINT#0;
    DataScanRecordCount := Producer.ScanRecordCount;
    SingleRecordOpsOk :=
        SingleRecordOpsOk AND
        (Producer.ScanRecordCount = UINT#1) AND
        (Producer.PublishedRecordCount - CountBefore = ULINT#1);
    OpsOk := OpsOk AND Producer.Done AND (NOT Producer.Error) AND (Producer.AssignedSeq = ULINT#0);
    Producer(Execute := FALSE, Op := UINT#0, SourceId := UDINT#30);

    CountBefore := Producer.PublishedRecordCount;
    Producer(Execute := TRUE, Op := UINT#0, SourceId := UDINT#10);
    SingleRecordOpsOk :=
        SingleRecordOpsOk AND
        (Producer.ScanRecordCount = UINT#1) AND
        (Producer.PublishedRecordCount - CountBefore = ULINT#1);
    OpsOk := OpsOk AND Producer.Done AND (NOT Producer.Error) AND (Producer.AssignedSeq = ULINT#0);
    Producer(Execute := FALSE, Op := UINT#0, SourceId := UDINT#10);

    CountBefore := Producer.PublishedRecordCount;
    Producer(
        Execute := TRUE,
        Op := UINT#1,
        DefHashOld := DefHashOld,
        DefHashNew := DefHashNew,
        TransitionEpochId := ULINT#2);
    BurstScanRecordCount := Producer.ScanRecordCount;
    BurstPublishedDelta := Producer.PublishedRecordCount - CountBefore;
    Offset0 := Producer.ScanRecordOffsets[0];
    Offset1 := Producer.ScanRecordOffsets[1];
    Offset2 := Producer.ScanRecordOffsets[2];
    Length0 := Producer.ScanRecordLengths[0];
    Length1 := Producer.ScanRecordLengths[1];
    Length2 := Producer.ScanRecordLengths[2];
    BurstBytes := Length0 + Length1 + Length2;
    BurstContiguousOk :=
        (BurstScanRecordCount = UINT#3) AND
        (BurstPublishedDelta = ULINT#3) AND
        (Offset0 = UINT#0) AND
        (Length0 = UINT#44) AND
        (Offset1 = Offset0 + Length0) AND
        (Length1 = UINT#56) AND
        (Offset2 = Offset1 + Length1) AND
        (Length2 = UINT#56) AND
        (BurstBytes = UINT#156);
    BurstCrcOk :=
        OPENOT_TestScanRecordCrcValid(
            Records := Producer.ScanRecords,
            Offset := Offset0,
            Length := Length0) AND
        OPENOT_TestScanRecordCrcValid(
            Records := Producer.ScanRecords,
            Offset := Offset1,
            Length := Length1) AND
        OPENOT_TestScanRecordCrcValid(
            Records := Producer.ScanRecords,
            Offset := Offset2,
            Length := Length2);
    BurstOrderOk :=
        OPENOT_TestScanRecordHeaderOk(
            Records := Producer.ScanRecords,
            Offset := Offset0,
            Length := Length0,
            EventTypeId := UDINT#16#0102,
            SourceId := UDINT#0) AND
        OPENOT_TestScanRecordHeaderOk(
            Records := Producer.ScanRecords,
            Offset := Offset1,
            Length := Length1,
            EventTypeId := UDINT#16#80000108,
            SourceId := UDINT#10) AND
        OPENOT_TestScanRecordHeaderOk(
            Records := Producer.ScanRecords,
            Offset := Offset2,
            Length := Length2,
            EventTypeId := UDINT#16#80000108,
            SourceId := UDINT#30);
    OpsOk := OpsOk AND Producer.Done AND (NOT Producer.Error) AND Producer.TransitionOpen;
    Producer(Execute := FALSE, Op := UINT#1);
    BurstNoEdgeScanRecordCount := Producer.ScanRecordCount;

    CountBefore := Producer.PublishedRecordCount;
    Producer(Execute := TRUE, Op := UINT#2);
    Delta := Producer.PublishedRecordCount - CountBefore;
    DefinitionChangedScanRecordCount := Producer.ScanRecordCount;
    SingleRecordOpsOk :=
        SingleRecordOpsOk AND
        (Producer.ScanRecordCount = UINT#1) AND
        (Delta = ULINT#1);
    OpsOk := OpsOk AND Producer.Done AND (NOT Producer.Error) AND Producer.DefinitionChangedEmitted;
    Producer(Execute := FALSE, Op := UINT#2);

    CountBefore := Producer.PublishedRecordCount;
    Producer(Execute := TRUE, Op := UINT#3);
    Delta := Producer.PublishedRecordCount - CountBefore;
    LoggerStartedScanRecordCount := Producer.ScanRecordCount;
    SingleRecordOpsOk :=
        SingleRecordOpsOk AND
        (Producer.ScanRecordCount = UINT#1) AND
        (Delta = ULINT#1);
    OpsOk :=
        OpsOk AND
        Producer.Done AND
        (NOT Producer.Error) AND
        (NOT Producer.TransitionOpen);
    Producer(Execute := FALSE, Op := UINT#3);

    CountBefore := Producer.PublishedRecordCount;
    Producer(Execute := TRUE, Checkpoint := TRUE, SourceId := UDINT#30);
    Delta := Producer.PublishedRecordCount - CountBefore;
    CheckpointScanRecordCount := Producer.ScanRecordCount;
    SingleRecordOpsOk :=
        SingleRecordOpsOk AND
        (Producer.ScanRecordCount = UINT#1) AND
        (Delta = ULINT#1);
    OpsOk := OpsOk AND Producer.Done AND Producer.CheckpointDone AND (NOT Producer.Error);
    Producer(Execute := FALSE, Checkpoint := TRUE, SourceId := UDINT#30);
    SingleNoEdgeScanRecordCount := Producer.ScanRecordCount;

    Ran := TRUE;
END_IF;

Passed :=
    OpsOk AND
    SingleRecordOpsOk AND
    BurstCrcOk AND
    BurstOrderOk AND
    BurstContiguousOk AND
    (BurstNoEdgeScanRecordCount = UINT#3) AND
    (SingleNoEdgeScanRecordCount = UINT#1) AND
    (Producer.PublishedRecordCount = ULINT#8) AND
    (Producer.EmissionCount = UINT#8);
END_FUNCTION_BLOCK

(* ---- test_source_high_water.st ---- *)
FUNCTION_BLOCK OPENOT_TestSourceHighWater
VAR_OUTPUT
    Passed : BOOL;
    MismatchIndex : UINT;
    ActualLength : UINT;
    ExpectedLength : UINT;
END_VAR
VAR
    Encoder : OPENOT_EncodeSourceHighWater;
    Expected : ARRAY[0..55] OF BYTE := [
        BYTE#16#4F, BYTE#16#4F, BYTE#16#54, BYTE#16#32, BYTE#16#38, BYTE#16#00, BYTE#16#08, BYTE#16#00,
        BYTE#16#00, BYTE#16#00, BYTE#16#00, BYTE#16#00, BYTE#16#00, BYTE#16#00, BYTE#16#00, BYTE#16#00,
        BYTE#16#01, BYTE#16#00, BYTE#16#00, BYTE#16#00, BYTE#16#00, BYTE#16#00, BYTE#16#00, BYTE#16#00,
        BYTE#16#05, BYTE#16#00, BYTE#16#00, BYTE#16#00, BYTE#16#00, BYTE#16#00, BYTE#16#00, BYTE#16#00,
        BYTE#16#58, BYTE#16#00, BYTE#16#00, BYTE#16#00, BYTE#16#08, BYTE#16#01, BYTE#16#00, BYTE#16#80,
        BYTE#16#38, BYTE#16#00, BYTE#16#07, BYTE#16#08, BYTE#16#05, BYTE#16#00, BYTE#16#00, BYTE#16#00,
        BYTE#16#00, BYTE#16#00, BYTE#16#00, BYTE#16#00, BYTE#16#CD, BYTE#16#D4, BYTE#16#74, BYTE#16#86
    ];
    Index : UINT;
END_VAR

Encoder(SourceId := UDINT#88, RunId := ULINT#1, ProducedCount := ULINT#5, SourceTime := ULINT#0);
ActualLength := Encoder.Length;
ExpectedLength := UINT#56;
Passed := ActualLength = ExpectedLength;
MismatchIndex := UINT#65535;

IF Passed THEN
    FOR Index := UINT#0 TO ExpectedLength - UINT#1 DO
        IF (Encoder.Buffer[Index] <> Expected[Index]) AND (MismatchIndex = UINT#65535) THEN
            Passed := FALSE;
            MismatchIndex := Index;
        END_IF;
    END_FOR;
END_IF;
END_FUNCTION_BLOCK

(* ---- test_transition_cold.st ---- *)
FUNCTION_BLOCK OPENOT_TestTransitionCold
VAR_OUTPUT
    Passed : BOOL;
    PostDataSeq : ULINT;
    SourceNextSeq : ULINT;
    SourceCountAfterColdData : UINT;
    EpochFirstAbsSet : BOOL;
    DefinitionHashOk : BOOL;
    PrevDefinitionHashOk : BOOL;
END_VAR
VAR
    Producer : OPENOT_Producer;
    DefHashOld : OPENOT_HASH8 := [
        BYTE#16#6F, BYTE#16#6C, BYTE#16#64, BYTE#16#68,
        BYTE#16#61, BYTE#16#73, BYTE#16#68, BYTE#16#31
    ];
    DefHashNew : OPENOT_HASH8 := [
        BYTE#16#6E, BYTE#16#65, BYTE#16#77, BYTE#16#68,
        BYTE#16#61, BYTE#16#73, BYTE#16#68, BYTE#16#32
    ];
    Ran : BOOL;
    OpsOk : BOOL;
    LogOk : BOOL;
    SourceFound : BOOL;
    HashIndex : UINT;
    SourceIndex : UINT;
END_VAR

IF NOT Ran THEN
    OpsOk := TRUE;

    Producer(Execute := TRUE, Op := UINT#0, SourceId := UDINT#21);
    OpsOk := OpsOk AND Producer.Done AND (NOT Producer.Error) AND (Producer.AssignedSeq = ULINT#0);
    Producer(Execute := FALSE, Op := UINT#0, SourceId := UDINT#21);

    Producer(
        Execute := TRUE,
        Op := UINT#1,
        DefHashOld := DefHashOld,
        DefHashNew := DefHashNew,
        TransitionEpochId := ULINT#2);
    OpsOk := OpsOk AND Producer.Done AND (NOT Producer.Error) AND Producer.TransitionOpen;
    Producer(Execute := FALSE, Op := UINT#1);

    Producer(Execute := TRUE, Op := UINT#2);
    OpsOk := OpsOk AND Producer.Done AND (NOT Producer.Error) AND Producer.DefinitionChangedEmitted;
    Producer(Execute := FALSE, Op := UINT#2);

    Producer(Execute := TRUE, Op := UINT#4);
    OpsOk :=
        OpsOk AND
        Producer.Done AND
        (NOT Producer.Error) AND
        (Producer.RunId = ULINT#2) AND
        (Producer.SystemSeq = ULINT#1) AND
        (Producer.SourceCount = UINT#0);
    Producer(Execute := FALSE, Op := UINT#4);

    Producer(Execute := TRUE, Op := UINT#0, SourceId := UDINT#21);
    PostDataSeq := Producer.AssignedSeq;
    OpsOk := OpsOk AND Producer.Done AND (NOT Producer.Error) AND (PostDataSeq = ULINT#0);

    Ran := TRUE;
END_IF;

SourceFound := FALSE;
SourceNextSeq := ULINT#0;
FOR SourceIndex := UINT#0 TO UINT#15 DO
    IF Producer.SourceUsed[SourceIndex] AND (Producer.SourceIds[SourceIndex] = UDINT#21) THEN
        SourceFound := TRUE;
        SourceNextSeq := Producer.SourceNextSeqs[SourceIndex];
    END_IF;
END_FOR;
SourceCountAfterColdData := Producer.SourceCount;

DefinitionHashOk := TRUE;
PrevDefinitionHashOk := TRUE;
FOR HashIndex := UINT#0 TO UINT#7 DO
    DefinitionHashOk := DefinitionHashOk AND (Producer.DefinitionHash[HashIndex] = DefHashNew[HashIndex]);
    PrevDefinitionHashOk := PrevDefinitionHashOk AND (Producer.PrevDefinitionHash[HashIndex] = DefHashOld[HashIndex]);
END_FOR;

EpochFirstAbsSet := Producer.EpochFirstAbs > ULINT#0;

LogOk :=
    (Producer.EmissionCount = UINT#6) AND
    (Producer.Emissions[0].EventTypeId = UDINT#16#0003) AND
    (Producer.Emissions[0].RunId = ULINT#1) AND
    (Producer.Emissions[0].SourceId = UDINT#21) AND
    (Producer.Emissions[0].Seq = ULINT#0) AND
    (Producer.Emissions[1].EventTypeId = UDINT#16#0102) AND
    (Producer.Emissions[1].RunId = ULINT#1) AND
    (Producer.Emissions[1].SourceId = UDINT#0) AND
    (Producer.Emissions[1].Seq = ULINT#0) AND
    (Producer.Emissions[2].EventTypeId = UDINT#16#80000108) AND
    (Producer.Emissions[2].RunId = ULINT#1) AND
    (Producer.Emissions[2].SourceId = UDINT#21) AND
    (Producer.Emissions[2].Seq = ULINT#1) AND
    (Producer.Emissions[3].EventTypeId = UDINT#16#0106) AND
    (Producer.Emissions[3].RunId = ULINT#1) AND
    (Producer.Emissions[3].SourceId = UDINT#0) AND
    (Producer.Emissions[3].Seq = ULINT#1) AND
    (Producer.Emissions[4].EventTypeId = UDINT#16#0101) AND
    (Producer.Emissions[4].RunId = ULINT#2) AND
    (Producer.Emissions[4].SourceId = UDINT#0) AND
    (Producer.Emissions[4].Seq = ULINT#0) AND
    (Producer.Emissions[5].EventTypeId = UDINT#16#0003) AND
    (Producer.Emissions[5].RunId = ULINT#2) AND
    (Producer.Emissions[5].SourceId = UDINT#21) AND
    (Producer.Emissions[5].Seq = ULINT#0);

Passed :=
    OpsOk AND
    LogOk AND
    SourceFound AND
    (SourceNextSeq = ULINT#1) AND
    (SourceCountAfterColdData = UINT#1) AND
    (Producer.PublishedRecordCount = ULINT#6) AND
    (Producer.RunId = ULINT#2) AND
    (Producer.EpochId = ULINT#2) AND
    (Producer.SystemSeq = ULINT#1) AND
    (Producer.SourceTime = ULINT#1780000000000000006) AND
    EpochFirstAbsSet AND
    DefinitionHashOk AND
    PrevDefinitionHashOk;
END_FUNCTION_BLOCK

(* ---- test_transition_guards.st ---- *)
FUNCTION_BLOCK OPENOT_TestTransitionGuards
VAR_OUTPUT
    Passed : BOOL;
    FinishBeforeDefinitionRejected : BOOL;
    DefinitionTwiceRejected : BOOL;
    BeginWhileOpenRejected : BOOL;
    FinishWithNoOpenRejected : BOOL;
    DefinitionWithNoOpenRejected : BOOL;
    CheckpointWhileOpenRejected : BOOL;
    HeldExecuteDidNotRepeat : BOOL;
END_VAR
VAR
    FinishProducer : OPENOT_Producer;
    TwiceProducer : OPENOT_Producer;
    OpenProducer : OPENOT_Producer;
    NoOpenProducer : OPENOT_Producer;
    CheckpointProducer : OPENOT_Producer;
    HeldProducer : OPENOT_Producer;
    DefHashOld : OPENOT_HASH8 := [
        BYTE#16#6F, BYTE#16#6C, BYTE#16#64, BYTE#16#68,
        BYTE#16#61, BYTE#16#73, BYTE#16#68, BYTE#16#31
    ];
    DefHashNew : OPENOT_HASH8 := [
        BYTE#16#6E, BYTE#16#65, BYTE#16#77, BYTE#16#68,
        BYTE#16#61, BYTE#16#73, BYTE#16#68, BYTE#16#32
    ];
    Ran : BOOL;
END_VAR

IF NOT Ran THEN
    FinishProducer(Execute := TRUE, Op := UINT#0, SourceId := UDINT#21);
    FinishProducer(Execute := FALSE, Op := UINT#0, SourceId := UDINT#21);
    FinishProducer(
        Execute := TRUE,
        Op := UINT#1,
        DefHashOld := DefHashOld,
        DefHashNew := DefHashNew,
        TransitionEpochId := ULINT#2);
    FinishProducer(Execute := FALSE, Op := UINT#1);
    FinishProducer(Execute := TRUE, Op := UINT#3);
    FinishBeforeDefinitionRejected := FinishProducer.Error AND (NOT FinishProducer.Done);

    TwiceProducer(
        Execute := TRUE,
        Op := UINT#1,
        DefHashOld := DefHashOld,
        DefHashNew := DefHashNew,
        TransitionEpochId := ULINT#2);
    TwiceProducer(Execute := FALSE, Op := UINT#1);
    TwiceProducer(Execute := TRUE, Op := UINT#2);
    TwiceProducer(Execute := FALSE, Op := UINT#2);
    TwiceProducer(Execute := TRUE, Op := UINT#2);
    DefinitionTwiceRejected := TwiceProducer.Error AND (NOT TwiceProducer.Done);

    OpenProducer(
        Execute := TRUE,
        Op := UINT#1,
        DefHashOld := DefHashOld,
        DefHashNew := DefHashNew,
        TransitionEpochId := ULINT#2);
    OpenProducer(Execute := FALSE, Op := UINT#1);
    OpenProducer(Execute := TRUE, Op := UINT#1);
    BeginWhileOpenRejected := OpenProducer.Error AND (NOT OpenProducer.Done);

    NoOpenProducer(Execute := TRUE, Op := UINT#3);
    FinishWithNoOpenRejected := NoOpenProducer.Error AND (NOT NoOpenProducer.Done);
    NoOpenProducer(Execute := FALSE, Op := UINT#3);
    NoOpenProducer(Execute := TRUE, Op := UINT#2);
    DefinitionWithNoOpenRejected := NoOpenProducer.Error AND (NOT NoOpenProducer.Done);

    CheckpointProducer(Execute := TRUE, Op := UINT#0, SourceId := UDINT#21);
    CheckpointProducer(Execute := FALSE, Op := UINT#0, SourceId := UDINT#21);
    CheckpointProducer(
        Execute := TRUE,
        Op := UINT#1,
        DefHashOld := DefHashOld,
        DefHashNew := DefHashNew,
        TransitionEpochId := ULINT#2);
    CheckpointProducer(Execute := FALSE, Op := UINT#1);
    CheckpointProducer(Execute := TRUE, SourceId := UDINT#21, Checkpoint := TRUE);
    CheckpointWhileOpenRejected := CheckpointProducer.Error AND (NOT CheckpointProducer.Done);

    HeldProducer(Execute := TRUE, Op := UINT#0, SourceId := UDINT#5);
    HeldProducer(Execute := TRUE, Op := UINT#0, SourceId := UDINT#5);
    HeldExecuteDidNotRepeat :=
        (HeldProducer.EmissionCount = UINT#1) AND
        (HeldProducer.SourceNextSeqs[0] = ULINT#1);

    Ran := TRUE;
END_IF;

Passed :=
    FinishBeforeDefinitionRejected AND
    DefinitionTwiceRejected AND
    BeginWhileOpenRejected AND
    FinishWithNoOpenRejected AND
    DefinitionWithNoOpenRejected AND
    CheckpointWhileOpenRejected AND
    HeldExecuteDidNotRepeat;
END_FUNCTION_BLOCK

(* ---- test_transition_high_water_order.st ---- *)
FUNCTION_BLOCK OPENOT_TestTransitionHighWaterOrder
VAR_OUTPUT
    Passed : BOOL;
    FirstHighWaterSource : UDINT;
    SecondHighWaterSource : UDINT;
END_VAR
VAR
    Producer : OPENOT_Producer;
    DefHashOld : OPENOT_HASH8 := [
        BYTE#16#6F, BYTE#16#6C, BYTE#16#64, BYTE#16#68,
        BYTE#16#61, BYTE#16#73, BYTE#16#68, BYTE#16#31
    ];
    DefHashNew : OPENOT_HASH8 := [
        BYTE#16#6E, BYTE#16#65, BYTE#16#77, BYTE#16#68,
        BYTE#16#61, BYTE#16#73, BYTE#16#68, BYTE#16#32
    ];
    Ran : BOOL;
    OpsOk : BOOL;
END_VAR

IF NOT Ran THEN
    OpsOk := TRUE;

    Producer(Execute := TRUE, Op := UINT#0, SourceId := UDINT#30);
    OpsOk := OpsOk AND Producer.Done AND (NOT Producer.Error);
    Producer(Execute := FALSE, Op := UINT#0, SourceId := UDINT#30);

    Producer(Execute := TRUE, Op := UINT#0, SourceId := UDINT#10);
    OpsOk := OpsOk AND Producer.Done AND (NOT Producer.Error);
    Producer(Execute := FALSE, Op := UINT#0, SourceId := UDINT#10);

    Producer(
        Execute := TRUE,
        Op := UINT#1,
        DefHashOld := DefHashOld,
        DefHashNew := DefHashNew,
        TransitionEpochId := ULINT#2);
    OpsOk := OpsOk AND Producer.Done AND (NOT Producer.Error);

    FirstHighWaterSource := Producer.Emissions[3].SourceId;
    SecondHighWaterSource := Producer.Emissions[4].SourceId;
    Ran := TRUE;
END_IF;

Passed :=
    OpsOk AND
    (Producer.EmissionCount = UINT#5) AND
    (Producer.PublishedRecordCount = ULINT#5) AND
    (Producer.Emissions[2].EventTypeId = UDINT#16#0102) AND
    (Producer.Emissions[3].EventTypeId = UDINT#16#80000108) AND
    (Producer.Emissions[3].SourceId = UDINT#10) AND
    (Producer.Emissions[3].Seq = ULINT#1) AND
    (Producer.Emissions[4].EventTypeId = UDINT#16#80000108) AND
    (Producer.Emissions[4].SourceId = UDINT#30) AND
    (Producer.Emissions[4].Seq = ULINT#1);
END_FUNCTION_BLOCK

(* ---- test_transition_warm.st ---- *)
FUNCTION_BLOCK OPENOT_TestTransitionWarm
VAR_OUTPUT
    Passed : BOOL;
    DataDuringTransitionRejected : BOOL;
    PostDataSeq : ULINT;
    SourceNextSeq : ULINT;
    EpochFirstAbsSet : BOOL;
    DefinitionHashOk : BOOL;
    PrevDefinitionHashOk : BOOL;
END_VAR
VAR
    Producer : OPENOT_Producer;
    DefHashOld : OPENOT_HASH8 := [
        BYTE#16#6F, BYTE#16#6C, BYTE#16#64, BYTE#16#68,
        BYTE#16#61, BYTE#16#73, BYTE#16#68, BYTE#16#31
    ];
    DefHashNew : OPENOT_HASH8 := [
        BYTE#16#6E, BYTE#16#65, BYTE#16#77, BYTE#16#68,
        BYTE#16#61, BYTE#16#73, BYTE#16#68, BYTE#16#32
    ];
    Ran : BOOL;
    OpsOk : BOOL;
    LogOk : BOOL;
    SourceFound : BOOL;
    HashIndex : UINT;
    SourceIndex : UINT;
    EmissionCountBeforeError : UINT;
END_VAR

IF NOT Ran THEN
    OpsOk := TRUE;

    Producer(Execute := TRUE, Op := UINT#0, SourceId := UDINT#21);
    OpsOk := OpsOk AND Producer.Done AND (NOT Producer.Error) AND (Producer.AssignedSeq = ULINT#0);
    Producer(Execute := FALSE, Op := UINT#0, SourceId := UDINT#21);

    Producer(Execute := TRUE, Op := UINT#0, SourceId := UDINT#21);
    OpsOk := OpsOk AND Producer.Done AND (NOT Producer.Error) AND (Producer.AssignedSeq = ULINT#1);
    Producer(Execute := FALSE, Op := UINT#0, SourceId := UDINT#21);

    Producer(
        Execute := TRUE,
        Op := UINT#1,
        DefHashOld := DefHashOld,
        DefHashNew := DefHashNew,
        TransitionEpochId := ULINT#2);
    OpsOk := OpsOk AND Producer.Done AND (NOT Producer.Error) AND Producer.TransitionOpen;
    EmissionCountBeforeError := Producer.EmissionCount;
    Producer(Execute := FALSE, Op := UINT#1);

    Producer(Execute := TRUE, Op := UINT#0, SourceId := UDINT#21);
    DataDuringTransitionRejected :=
        Producer.Error AND
        (NOT Producer.Done) AND
        (Producer.EmissionCount = EmissionCountBeforeError);
    Producer(Execute := FALSE, Op := UINT#0, SourceId := UDINT#21);

    Producer(Execute := TRUE, Op := UINT#2);
    OpsOk := OpsOk AND Producer.Done AND (NOT Producer.Error) AND Producer.DefinitionChangedEmitted;
    Producer(Execute := FALSE, Op := UINT#2);

    Producer(Execute := TRUE, Op := UINT#3);
    OpsOk :=
        OpsOk AND
        Producer.Done AND
        (NOT Producer.Error) AND
        (NOT Producer.TransitionOpen) AND
        (Producer.RunId = ULINT#1) AND
        (Producer.EpochId = ULINT#2);
    Producer(Execute := FALSE, Op := UINT#3);

    Producer(Execute := TRUE, Op := UINT#0, SourceId := UDINT#21);
    PostDataSeq := Producer.AssignedSeq;
    OpsOk := OpsOk AND Producer.Done AND (NOT Producer.Error) AND (PostDataSeq = ULINT#3);

    Ran := TRUE;
END_IF;

SourceFound := FALSE;
SourceNextSeq := ULINT#0;
FOR SourceIndex := UINT#0 TO UINT#15 DO
    IF Producer.SourceUsed[SourceIndex] AND (Producer.SourceIds[SourceIndex] = UDINT#21) THEN
        SourceFound := TRUE;
        SourceNextSeq := Producer.SourceNextSeqs[SourceIndex];
    END_IF;
END_FOR;

DefinitionHashOk := TRUE;
PrevDefinitionHashOk := TRUE;
FOR HashIndex := UINT#0 TO UINT#7 DO
    DefinitionHashOk := DefinitionHashOk AND (Producer.DefinitionHash[HashIndex] = DefHashNew[HashIndex]);
    PrevDefinitionHashOk := PrevDefinitionHashOk AND (Producer.PrevDefinitionHash[HashIndex] = DefHashOld[HashIndex]);
END_FOR;

EpochFirstAbsSet := Producer.EpochFirstAbs > ULINT#0;

LogOk :=
    (Producer.EmissionCount = UINT#7) AND
    (Producer.Emissions[0].EventTypeId = UDINT#16#0003) AND
    (Producer.Emissions[0].RunId = ULINT#1) AND
    (Producer.Emissions[0].SourceId = UDINT#21) AND
    (Producer.Emissions[0].Seq = ULINT#0) AND
    (Producer.Emissions[1].EventTypeId = UDINT#16#0003) AND
    (Producer.Emissions[1].RunId = ULINT#1) AND
    (Producer.Emissions[1].SourceId = UDINT#21) AND
    (Producer.Emissions[1].Seq = ULINT#1) AND
    (Producer.Emissions[2].EventTypeId = UDINT#16#0102) AND
    (Producer.Emissions[2].RunId = ULINT#1) AND
    (Producer.Emissions[2].SourceId = UDINT#0) AND
    (Producer.Emissions[2].Seq = ULINT#0) AND
    (Producer.Emissions[3].EventTypeId = UDINT#16#80000108) AND
    (Producer.Emissions[3].RunId = ULINT#1) AND
    (Producer.Emissions[3].SourceId = UDINT#21) AND
    (Producer.Emissions[3].Seq = ULINT#2) AND
    (Producer.Emissions[4].EventTypeId = UDINT#16#0106) AND
    (Producer.Emissions[4].RunId = ULINT#1) AND
    (Producer.Emissions[4].SourceId = UDINT#0) AND
    (Producer.Emissions[4].Seq = ULINT#1) AND
    (Producer.Emissions[5].EventTypeId = UDINT#16#0101) AND
    (Producer.Emissions[5].RunId = ULINT#1) AND
    (Producer.Emissions[5].SourceId = UDINT#0) AND
    (Producer.Emissions[5].Seq = ULINT#2) AND
    (Producer.Emissions[6].EventTypeId = UDINT#16#0003) AND
    (Producer.Emissions[6].RunId = ULINT#1) AND
    (Producer.Emissions[6].SourceId = UDINT#21) AND
    (Producer.Emissions[6].Seq = ULINT#3);

Passed :=
    OpsOk AND
    DataDuringTransitionRejected AND
    LogOk AND
    SourceFound AND
    (Producer.PublishedRecordCount = ULINT#7) AND
    (SourceNextSeq = ULINT#4) AND
    (Producer.SourceTime = ULINT#1780000000000000007) AND
    EpochFirstAbsSet AND
    DefinitionHashOk AND
    PrevDefinitionHashOk;
END_FUNCTION_BLOCK
